LIN {X 0,Y 476.312,Z 880.73,A -85,B 0,C 180,E1 -14353.297,E2 -14353.297} C_VEL
LIN {X 0,Y 480.673,Z 862.161,A -85,B 0,C 180,E1 -14354.593,E2 -14354.593} C_VEL
LIN {X 0,Y 485.784,Z 837.994,A -85,B 0,C 180,E1 -14356.003,E2 -14356.003} C_VEL
LIN {X 0,Y 489.516,Z 817.506,A -85,B 0,C 180,E1 -14356.992,E2 -14356.992} C_VEL
LIN {X 0,Y 493.406,Z 792.396,A -85,B 0,C 180,E1 -14357.969,E2 -14357.969} C_VEL
LIN {X 0,Y 496.099,Z 770.51,A -85,B 0,C 180,E1 -14358.628,E2 -14358.628} C_VEL
LIN {X 0,Y 498.452,Z 745.206,A -85,B 0,C 180,E1 -14359.196,E2 -14359.196} C_VEL
LIN {X 0,Y 501.921,Z 674.53,A -85,B 0,C 180,E1 -14360.305,E2 -14360.305} C_VEL
LIN {X 0,Y 511.78,Z 467.818,A -85,B 0,C 180,E1 -14363.486,E2 -14363.486} C_VEL
LIN {X 0,Y 504.78,Z 456.576,A -85,B 0,C 180,E1 -14364.8,E2 -14364.8} C_VEL
LIN {X 0,Y 492.925,Z 439.35,A -85,B 0,C 180,E1 -14367.172,E2 -14367.172} C_VEL
LIN {X 0,Y 482.888,Z 425.653,A -85,B 0,C 180,E1 -14369.377,E2 -14369.377} C_VEL
LIN {X 0,Y 474.182,Z 414.504,A -85,B 0,C 180,E1 -14371.47,E2 -14371.47} C_VEL
LIN {X 0,Y 470.031,Z 409.325,A -85,B 0,C 180,E1 -14372.542,E2 -14372.542} C_VEL
LIN {X 0,Y 465.619,Z 403.891,A -85,B 0,C 180,E1 -14373.744,E2 -14373.744} C_VEL
LIN {X 0,Y 461.89,Z 399.125,A -85,B 0,C 180,E1 -14374.825,E2 -14374.825} C_VEL
LIN {X 0,Y 457.865,Z 394.726,A -85,B 0,C 180,E1 -14376.034,E2 -14376.034} C_VEL
LIN {X 0,Y 456.425,Z 392.715,A -85,B 0,C 180,E1 -14376.502,E2 -14376.502} C_VEL
LIN {X 0,Y 452.979,Z 389.244,A -85,B 0,C 180,E1 -14377.618,E2 -14377.618} C_VEL
LIN {X 0,Y 451.321,Z 386.663,A -85,B 0,C 180,E1 -14378.217,E2 -14378.217} C_VEL
LIN {X 0,Y 447.983,Z 383.799,A -85,B 0,C 180,E1 -14379.384,E2 -14379.384} C_VEL
LIN {X 0,Y 445.946,Z 380.402,A -85,B 0,C 180,E1 -14380.21,E2 -14380.21} C_VEL
LIN {X 0,Y 442.622,Z 378.058,A -85,B 0,C 180,E1 -14381.495,E2 -14381.495} C_VEL
LIN {X 0,Y 440.723,Z 374.852,A -85,B 0,C 180,E1 -14382.369,E2 -14382.369} C_VEL
LIN {X 0,Y 440.365,Z 373.869,A -85,B 0,C 180,E1 -14382.559,E2 -14382.559} C_VEL
LIN {X 0,Y 437.089,Z 372.153,A -85,B 0,C 180,E1 -14383.999,E2 -14383.999} C_VEL
LIN {X 0,Y 435.021,Z 369.435,A -85,B 0,C 180,E1 -14385.082,E2 -14385.082} C_VEL
LIN {X 0,Y 434.375,Z 367.098,A -85,B 0,C 180,E1 -14385.537,E2 -14385.537} C_VEL
LIN {X 0,Y 434.364,Z 367.103,A -85,B 0,C 180,E1 -14389.254,E2 -14389.254} C_VEL
LIN {X 0,Y 434.366,Z 367.111,A -85,B 0,C 180,E1 -14392.992,E2 -14392.992} C_VEL
LIN {X 0,Y 434.383,Z 367.122,A -85,B 0,C 180,E1 -14396.701,E2 -14396.701} C_VEL
LIN {X 0,Y 434.418,Z 367.114,A -85,B 0,C 180,E1 -14400.396,E2 -14400.396} C_VEL
LIN {X 0,Y 434.401,Z 367.104,A -85,B 0,C 180,E1 -14404.224,E2 -14404.224} C_VEL
LIN {X 0,Y 434.377,Z 367.098,A -85,B 0,C 180,E1 -14407.939,E2 -14407.939} C_VEL
LIN {X 0,Y 434.362,Z 367.095,A -85,B 0,C 180,E1 -14411.688,E2 -14411.688} C_VEL
LIN {X 0,Y 434.36,Z 367.094,A -85,B 0,C 180,E1 -14415.488,E2 -14415.488} C_VEL
LIN {X 0,Y 434.417,Z 367.337,A -85,B 0,C 180,E1 -14416.171,E2 -14416.171} C_VEL
LIN {X 0,Y 435.494,Z 370.263,A -85,B 0,C 180,E1 -14416.85,E2 -14416.85} C_VEL
LIN {X 0,Y 437.713,Z 372.671,A -85,B 0,C 180,E1 -14417.962,E2 -14417.962} C_VEL
LIN {X 0,Y 440.378,Z 374.005,A -85,B 0,C 180,E1 -14419.119,E2 -14419.119} C_VEL
LIN {X 0,Y 442.007,Z 377.269,A -85,B 0,C 180,E1 -14419.905,E2 -14419.905} C_VEL
LIN {X 0,Y 445.233,Z 380.091,A -85,B 0,C 180,E1 -14421.197,E2 -14421.197} C_VEL
LIN {X 0,Y 446.288,Z 380.829,A -85,B 0,C 180,E1 -14421.591,E2 -14421.591} C_VEL
LIN {X 0,Y 448.678,Z 384.586,A -85,B 0,C 180,E1 -14422.539,E2 -14422.539} C_VEL
LIN {X 0,Y 451.531,Z 387.353,A -85,B 0,C 180,E1 -14423.54,E2 -14423.54} C_VEL
LIN {X 0,Y 459.737,Z 397.67,A -85,B 0,C 180,E1 -14426.235,E2 -14426.235} C_VEL
LIN {X 0,Y 464.655,Z 404.165,A -85,B 0,C 180,E1 -14427.698,E2 -14427.698} C_VEL
LIN {X 0,Y 471.602,Z 413.51,A -85,B 0,C 180,E1 -14429.604,E2 -14429.604} C_VEL
LIN {X 0,Y 481.089,Z 426.79,A -85,B 0,C 180,E1 -14431.97,E2 -14431.97} C_VEL
LIN {X 0,Y 492.017,Z 443.215,A -85,B 0,C 180,E1 -14434.435,E2 -14434.435} C_VEL
LIN {X 0,Y 503.274,Z 461.442,A -85,B 0,C 180,E1 -14436.746,E2 -14436.746} C_VEL
LIN {X 0,Y 511.643,Z 476.212,A -85,B 0,C 180,E1 -14438.349,E2 -14438.349} C_VEL
LIN {X 0,Y 499.968,Z 722.479,A -85,B 0,C 180,E1 -14442.13,E2 -14442.13} C_VEL
LIN {X 0,Y 497.691,Z 766.294,A -85,B 0,C 180,E1 -14442.836,E2 -14442.836} C_VEL
LIN {X 0,Y 495.246,Z 790.201,A -85,B 0,C 180,E1 -14443.379,E2 -14443.379} C_VEL
LIN {X 0,Y 492.423,Z 811.739,A -85,B 0,C 180,E1 -14444.014,E2 -14444.014} C_VEL
LIN {X 0,Y 488.567,Z 835.485,A -85,B 0,C 180,E1 -14444.918,E2 -14444.918} C_VEL
LIN {X 0,Y 484.947,Z 854.788,A -85,B 0,C 180,E1 -14445.821,E2 -14445.821} C_VEL
LIN {X 0,Y 480.203,Z 877.436,A -85,B 0,C 180,E1 -14447.087,E2 -14447.087} C_VEL
LIN {X 0,Y 475.462,Z 897.422,A -85,B 0,C 180,E1 -14448.433,E2 -14448.433} C_VEL
LIN {X 0,Y 470.467,Z 917.266,A -85,B 0,C 180,E1 -14449.991,E2 -14449.991} C_VEL
LIN {X 0,Y 464.895,Z 937.64,A -85,B 0,C 180,E1 -14451.883,E2 -14451.883} C_VEL
LIN {X 0,Y 459.973,Z 955.021,A -85,B 0,C 180,E1 -14453.754,E2 -14453.754} C_VEL
LIN {X 0,Y 454.665,Z 973.247,A -85,B 0,C 180,E1 -14456.042,E2 -14456.042} C_VEL
LIN {X 0,Y 450.242,Z 988.386,A -85,B 0,C 180,E1 -14458.242,E2 -14458.242} C_VEL
LIN {X 0,Y 445.524,Z 1004.762,A -85,B 0,C 180,E1 -14461.003,E2 -14461.003} C_VEL
LIN {X 0,Y 441.972,Z 1017.607,A -85,B 0,C 180,E1 -14463.533,E2 -14463.533} C_VEL
LIN {X 0,Y 438.648,Z 1030.56,A -85,B 0,C 180,E1 -14466.49,E2 -14466.49} C_VEL
LIN {X 0,Y 436.221,Z 1041.033,A -85,B 0,C 180,E1 -14469.33,E2 -14469.33} C_VEL
LIN {X 0,Y 434.319,Z 1050.833,A -85,B 0,C 180,E1 -14472.447,E2 -14472.447} C_VEL
LIN {X 0,Y 433.067,Z 1058.69,A -85,B 0,C 180,E1 -14475.561,E2 -14475.561} C_VEL
LIN {X 0,Y 432.375,Z 1064.792,A -85,B 0,C 180,E1 -14478.529,E2 -14478.529} C_VEL
LIN {X 0,Y 432.028,Z 1069.722,A -85,B 0,C 180,E1 -14481.75,E2 -14481.75} C_VEL
LIN {X 0,Y 431.948,Z 1072.642,A -85,B 0,C 180,E1 -14484.494,E2 -14484.494} C_VEL
LIN {X 0,Y 431.942,Z 1074.478,A -85,B 0,C 180,E1 -14487.346,E2 -14487.346} C_VEL
LIN {X 0,Y 431.944,Z 1074.935,A -85,B 0,C 180,E1 -14490.531,E2 -14490.531} C_VEL
LIN {X 0,Y 431.947,Z 1074.097,A -85,B 0,C 180,E1 -14493.185,E2 -14493.185} C_VEL
LIN {X 0,Y 431.957,Z 1072.052,A -85,B 0,C 180,E1 -14495.979,E2 -14495.979} C_VEL
LIN {X 0,Y 432.098,Z 1067.939,A -85,B 0,C 180,E1 -14499.322,E2 -14499.322} C_VEL
LIN {X 0,Y 432.468,Z 1063.258,A -85,B 0,C 180,E1 -14502.039,E2 -14502.039} C_VEL
LIN {X 0,Y 433.263,Z 1056.581,A -85,B 0,C 180,E1 -14505.116,E2 -14505.116} C_VEL
LIN {X 0,Y 434.613,Z 1047.978,A -85,B 0,C 180,E1 -14508.233,E2 -14508.233} C_VEL
LIN {X 0,Y 436.447,Z 1038.639,A -85,B 0,C 180,E1 -14511.081,E2 -14511.081} C_VEL
LIN {X 0,Y 439.195,Z 1026.418,A -85,B 0,C 180,E1 -14514.192,E2 -14514.192} C_VEL
LIN {X 0,Y 442.123,Z 1014.703,A -85,B 0,C 180,E1 -14516.747,E2 -14516.747} C_VEL
LIN {X 0,Y 446.307,Z 998.982,A -85,B 0,C 180,E1 -14519.678,E2 -14519.678} C_VEL
LIN {X 0,Y 450.249,Z 984.69,A -85,B 0,C 180,E1 -14521.969,E2 -14521.969} C_VEL
LIN {X 0,Y 455.37,Z 966.303,A -85,B 0,C 180,E1 -14524.507,E2 -14524.507} C_VEL
LIN {X 0,Y 459.837,Z 950.082,A -85,B 0,C 180,E1 -14526.433,E2 -14526.433} C_VEL
LIN {X 0,Y 465.189,Z 930.126,A -85,B 0,C 180,E1 -14528.481,E2 -14528.481} C_VEL
LIN {X 0,Y 469.751,Z 912.077,A -85,B 0,C 180,E1 -14530.063,E2 -14530.063} C_VEL
LIN {X 0,Y 474.735,Z 891.264,A -85,B 0,C 180,E1 -14531.645,E2 -14531.645} C_VEL
LIN {X 0,Y 479.385,Z 869.689,A -85,B 0,C 180,E1 -14533.004,E2 -14533.004} C_VEL
LIN {X 0,Y 483.602,Z 848.094,A -85,B 0,C 180,E1 -14534.155,E2 -14534.155} C_VEL
LIN {X 0,Y 487.514,Z 824.79,A -85,B 0,C 180,E1 -14535.16,E2 -14535.16} C_VEL
LIN {X 0,Y 490.647,Z 802.953,A -85,B 0,C 180,E1 -14535.914,E2 -14535.914} C_VEL
LIN {X 0,Y 493.595,Z 776.73,A -85,B 0,C 180,E1 -14536.597,E2 -14536.597} C_VEL
LIN {X 0,Y 495.266,Z 754.369,A -85,B 0,C 180,E1 -14537.023,E2 -14537.023} C_VEL
LIN {X 0,Y 506.388,Z 505.867,A -85,B 0,C 180,E1 -14540.839,E2 -14540.839} C_VEL
LIN {X 0,Y 507.752,Z 473.861,A -85,B 0,C 180,E1 -14541.346,E2 -14541.346} C_VEL
LIN {X 0,Y 496.766,Z 454.506,A -85,B 0,C 180,E1 -14543.341,E2 -14543.341} C_VEL
LIN {X 0,Y 485.526,Z 436.238,A -85,B 0,C 180,E1 -14545.541,E2 -14545.541} C_VEL
LIN {X 0,Y 474.396,Z 419.479,A -85,B 0,C 180,E1 -14547.917,E2 -14547.917} C_VEL
LIN {X 0,Y 464.351,Z 405.315,A -85,B 0,C 180,E1 -14550.277,E2 -14550.277} C_VEL
LIN {X 0,Y 456.195,Z 394.492,A -85,B 0,C 180,E1 -14552.382,E2 -14552.382} C_VEL
LIN {X 0,Y 451.654,Z 388.602,A -85,B 0,C 180,E1 -14553.648,E2 -14553.648} C_VEL
LIN {X 0,Y 448.444,Z 384.751,A -85,B 0,C 180,E1 -14554.582,E2 -14554.582} C_VEL
LIN {X 0,Y 444.619,Z 379.774,A -85,B 0,C 180,E1 -14555.769,E2 -14555.769} C_VEL
LIN {X 0,Y 441.559,Z 377.023,A -85,B 0,C 180,E1 -14556.725,E2 -14556.725} C_VEL
LIN {X 0,Y 439.696,Z 373.645,A -85,B 0,C 180,E1 -14557.399,E2 -14557.399} C_VEL
LIN {X 0,Y 436.563,Z 371.7,A -85,B 0,C 180,E1 -14558.432,E2 -14558.432} C_VEL
LIN {X 0,Y 434.835,Z 368.902,A -85,B 0,C 180,E1 -14559.102,E2 -14559.102} C_VEL
LIN {X 0,Y 434.414,Z 367.107,A -85,B 0,C 180,E1 -14559.345,E2 -14559.345} C_VEL
LIN {X 0,Y 434.406,Z 367.12,A -85,B 0,C 180,E1 -14563.241,E2 -14563.241} C_VEL
LIN {X 0,Y 434.37,Z 367.098,A -85,B 0,C 180,E1 -14566.835,E2 -14566.835} C_VEL
LIN {X 0,Y 434.36,Z 367.086,A -85,B 0,C 180,E1 -14570.593,E2 -14570.593} C_VEL
LIN {X 0,Y 434.362,Z 367.096,A -85,B 0,C 180,E1 -14574.452,E2 -14574.452} C_VEL
LIN {X 0,Y 434.383,Z 367.125,A -85,B 0,C 180,E1 -14578.153,E2 -14578.153} C_VEL
LIN {X 0,Y 434.41,Z 367.084,A -85,B 0,C 180,E1 -14581.715,E2 -14581.715} C_VEL
LIN {X 0,Y 434.396,Z 367.082,A -85,B 0,C 180,E1 -14585.548,E2 -14585.548} C_VEL
LIN {X 0,Y 434.37,Z 367.117,A -85,B 0,C 180,E1 -14589.139,E2 -14589.139} C_VEL
LIN {X 0,Y 434.365,Z 367.108,A -85,B 0,C 180,E1 -14592.902,E2 -14592.902} C_VEL
LIN {X 0,Y 434.373,Z 367.087,A -85,B 0,C 180,E1 -14596.585,E2 -14596.585} C_VEL
LIN {X 0,Y 434.407,Z 367.088,A -85,B 0,C 180,E1 -14600.198,E2 -14600.198} C_VEL
LIN {X 0,Y 434.403,Z 367.369,A -85,B 0,C 180,E1 -14603.107,E2 -14603.107} C_VEL
LIN {X 0,Y 435.405,Z 370.151,A -85,B 0,C 180,E1 -14603.552,E2 -14603.552} C_VEL
LIN {X 0,Y 438.005,Z 372.837,A -85,B 0,C 180,E1 -14604.478,E2 -14604.478} C_VEL
LIN {X 0,Y 440.013,Z 374.076,A -85,B 0,C 180,E1 -14605.129,E2 -14605.129} C_VEL
LIN {X 0,Y 442.037,Z 377.566,A -85,B 0,C 180,E1 -14605.849,E2 -14605.849} C_VEL
LIN {X 0,Y 445.524,Z 380.607,A -85,B 0,C 180,E1 -14606.923,E2 -14606.923} C_VEL
LIN {X 0,Y 448.383,Z 384.646,A -85,B 0,C 180,E1 -14607.816,E2 -14607.816} C_VEL
LIN {X 0,Y 450.75,Z 386.798,A -85,B 0,C 180,E1 -14608.485,E2 -14608.485} C_VEL
LIN {X 0,Y 454.01,Z 391.044,A -85,B 0,C 180,E1 -14609.415,E2 -14609.415} C_VEL
LIN {X 0,Y 455.822,Z 392.993,A -85,B 0,C 180,E1 -14609.901,E2 -14609.901} C_VEL
LIN {X 0,Y 459.596,Z 397.562,A -85,B 0,C 180,E1 -14610.893,E2 -14610.893} C_VEL
LIN {X 0,Y 465.963,Z 405.657,A -85,B 0,C 180,E1 -14612.48,E2 -14612.48} C_VEL
LIN {X 0,Y 473.123,Z 414.677,A -85,B 0,C 180,E1 -14614.132,E2 -14614.132} C_VEL
LIN {X 0,Y 484.592,Z 430.179,A -85,B 0,C 180,E1 -14616.57,E2 -14616.57} C_VEL
LIN {X 0,Y 496.643,Z 447.502,A -85,B 0,C 180,E1 -14618.895,E2 -14618.895} C_VEL
LIN {X 0,Y 506.73,Z 463.438,A -85,B 0,C 180,E1 -14620.704,E2 -14620.704} C_VEL
LIN {X 0,Y 508.051,Z 466.028,A -85,B 0,C 180,E1 -14620.942,E2 -14620.942} C_VEL
LIN {X 0,Y 496.67,Z 717.844,A -85,B 0,C 180,E1 -14624.797,E2 -14624.797} C_VEL
LIN {X 0,Y 494.808,Z 751.173,A -85,B 0,C 180,E1 -14625.359,E2 -14625.359} C_VEL
LIN {X 0,Y 492.684,Z 773.474,A -85,B 0,C 180,E1 -14625.895,E2 -14625.895} C_VEL
LIN {X 0,Y 489.778,Z 797.274,A -85,B 0,C 180,E1 -14626.645,E2 -14626.645} C_VEL
LIN {X 0,Y 486.432,Z 818.959,A -85,B 0,C 180,E1 -14627.526,E2 -14627.526} C_VEL
LIN {X 0,Y 482.523,Z 841.197,A -85,B 0,C 180,E1 -14628.621,E2 -14628.621} C_VEL
LIN {X 0,Y 478.106,Z 862.578,A -85,B 0,C 180,E1 -14629.899,E2 -14629.899} C_VEL
LIN {X 0,Y 473.753,Z 881.913,A -85,B 0,C 180,E1 -14631.26,E2 -14631.26} C_VEL
LIN {X 0,Y 468.395,Z 903.636,A -85,B 0,C 180,E1 -14633.064,E2 -14633.064} C_VEL
LIN {X 0,Y 463.901,Z 920.654,A -85,B 0,C 180,E1 -14634.715,E2 -14634.715} C_VEL
LIN {X 0,Y 458.704,Z 939.537,A -85,B 0,C 180,E1 -14636.83,E2 -14636.83} C_VEL
LIN {X 0,Y 453.988,Z 955.906,A -85,B 0,C 180,E1 -14638.978,E2 -14638.978} C_VEL
LIN {X 0,Y 449.39,Z 972.081,A -85,B 0,C 180,E1 -14641.421,E2 -14641.421} C_VEL
LIN {X 0,Y 445.178,Z 986.714,A -85,B 0,C 180,E1 -14644.025,E2 -14644.025} C_VEL
LIN {X 0,Y 441.519,Z 1000.18,A -85,B 0,C 180,E1 -14646.793,E2 -14646.793} C_VEL
LIN {X 0,Y 438.535,Z 1011.589,A -85,B 0,C 180,E1 -14649.583,E2 -14649.583} C_VEL
LIN {X 0,Y 436.196,Z 1021.758,A -85,B 0,C 180,E1 -14652.478,E2 -14652.478} C_VEL
LIN {X 0,Y 434.361,Z 1030.763,A -85,B 0,C 180,E1 -14655.605,E2 -14655.605} C_VEL
LIN {X 0,Y 433.253,Z 1037.454,A -85,B 0,C 180,E1 -14658.417,E2 -14658.417} C_VEL
LIN {X 0,Y 432.461,Z 1043.675,A -85,B 0,C 180,E1 -14661.758,E2 -14661.758} C_VEL
LIN {X 0,Y 432.383,Z 1044.478,A -85,B 0,C 180,E1 -14662.289,E2 -14662.289} C_VEL
LIN {X 0,Y 431.252,Z 1046.049,A -85,B 0,C 180,E1 -14663.288,E2 -14663.288} C_VEL
LIN {X 0,Y 424.68,Z 1049.373,A -85,B 0,C 180,E1 -14666.043,E2 -14666.043} C_VEL
LIN {X 0,Y 424.015,Z 1050.046,A -85,B 0,C 180,E1 -14666.861,E2 -14666.861} C_VEL
LIN {X 0,Y 423.97,Z 1051.839,A -85,B 0,C 180,E1 -14670,E2 -14670} C_VEL
LIN {X 0,Y 423.952,Z 1052.046,A -85,B 0,C 180,E1 -14673.11,E2 -14673.11} C_VEL
LIN {X 0,Y 423.99,Z 1051.15,A -85,B 0,C 180,E1 -14675.82,E2 -14675.82} C_VEL
LIN {X 0,Y 424.116,Z 1048.864,A -85,B 0,C 180,E1 -14678.952,E2 -14678.952} C_VEL
LIN {X 0,Y 424.471,Z 1044.87,A -85,B 0,C 180,E1 -14682.154,E2 -14682.154} C_VEL
LIN {X 0,Y 425.153,Z 1039.888,A -85,B 0,C 180,E1 -14685.133,E2 -14685.133} C_VEL
LIN {X 0,Y 426.447,Z 1032.657,A -85,B 0,C 180,E1 -14688.453,E2 -14688.453} C_VEL
LIN {X 0,Y 428.084,Z 1025.127,A -85,B 0,C 180,E1 -14691.257,E2 -14691.257} C_VEL
LIN {X 0,Y 430.657,Z 1015.015,A -85,B 0,C 180,E1 -14694.411,E2 -14694.411} C_VEL
LIN {X 0,Y 433.776,Z 1003.834,A -85,B 0,C 180,E1 -14697.304,E2 -14697.304} C_VEL
LIN {X 0,Y 437.683,Z 990.946,A -85,B 0,C 180,E1 -14700.172,E2 -14700.172} C_VEL
LIN {X 0,Y 441.9,Z 977.282,A -85,B 0,C 180,E1 -14702.737,E2 -14702.737} C_VEL
LIN {X 0,Y 446.55,Z 962.651,A -85,B 0,C 180,E1 -14705.132,E2 -14705.132} C_VEL
LIN {X 0,Y 451.957,Z 945.292,A -85,B 0,C 180,E1 -14707.554,E2 -14707.554} C_VEL
LIN {X 0,Y 457.023,Z 928.778,A -85,B 0,C 180,E1 -14709.543,E2 -14709.543} C_VEL
LIN {X 0,Y 462.732,Z 909.231,A -85,B 0,C 180,E1 -14711.558,E2 -14711.558} C_VEL
LIN {X 0,Y 467.522,Z 891.777,A -85,B 0,C 180,E1 -14713.103,E2 -14713.103} C_VEL
LIN {X 0,Y 472.813,Z 871.108,A -85,B 0,C 180,E1 -14714.681,E2 -14714.681} C_VEL
LIN {X 0,Y 477.553,Z 850.328,A -85,B 0,C 180,E1 -14716.004,E2 -14716.004} C_VEL
LIN {X 0,Y 481.999,Z 828.767,A -85,B 0,C 180,E1 -14717.166,E2 -14717.166} C_VEL
LIN {X 0,Y 485.904,Z 806.181,A -85,B 0,C 180,E1 -14718.152,E2 -14718.152} C_VEL
LIN {X 0,Y 488.82,Z 786.379,A -85,B 0,C 180,E1 -14718.857,E2 -14718.857} C_VEL
LIN {X 0,Y 491.753,Z 761.453,A -85,B 0,C 180,E1 -14719.548,E2 -14719.548} C_VEL
LIN {X 0,Y 493.545,Z 739.017,A -85,B 0,C 180,E1 -14719.998,E2 -14719.998} C_VEL
LIN {X 0,Y 505.635,Z 494.649,A -85,B 0,C 180,E1 -14723.782,E2 -14723.782} C_VEL
LIN {X 0,Y 506.705,Z 471.513,A -85,B 0,C 180,E1 -14724.156,E2 -14724.156} C_VEL
LIN {X 0,Y 496.592,Z 455.764,A -85,B 0,C 180,E1 -14726.135,E2 -14726.135} C_VEL
LIN {X 0,Y 485.373,Z 439.786,A -85,B 0,C 180,E1 -14728.518,E2 -14728.518} C_VEL
LIN {X 0,Y 475.719,Z 426.782,A -85,B 0,C 180,E1 -14730.78,E2 -14730.78} C_VEL
LIN {X 0,Y 467.493,Z 416.348,A -85,B 0,C 180,E1 -14732.898,E2 -14732.898} C_VEL
LIN {X 0,Y 463.038,Z 410.841,A -85,B 0,C 180,E1 -14734.138,E2 -14734.138} C_VEL
LIN {X 0,Y 458.779,Z 405.565,A -85,B 0,C 180,E1 -14735.4,E2 -14735.4} C_VEL
LIN {X 0,Y 455.074,Z 401.044,A -85,B 0,C 180,E1 -14736.566,E2 -14736.566} C_VEL
LIN {X 0,Y 450.464,Z 395.877,A -85,B 0,C 180,E1 -14738.105,E2 -14738.105} C_VEL
LIN {X 0,Y 449.141,Z 394.029,A -85,B 0,C 180,E1 -14738.586,E2 -14738.586} C_VEL
LIN {X 0,Y 445.811,Z 390.841,A -85,B 0,C 180,E1 -14739.794,E2 -14739.794} C_VEL
LIN {X 0,Y 444.018,Z 387.983,A -85,B 0,C 180,E1 -14740.532,E2 -14740.532} C_VEL
LIN {X 0,Y 440.775,Z 385.427,A -85,B 0,C 180,E1 -14741.825,E2 -14741.825} C_VEL
LIN {X 0,Y 438.663,Z 381.728,A -85,B 0,C 180,E1 -14742.831,E2 -14742.831} C_VEL
LIN {X 0,Y 434.968,Z 379.222,A -85,B 0,C 180,E1 -14744.534,E2 -14744.534} C_VEL
LIN {X 0,Y 433.08,Z 376.196,A -85,B 0,C 180,E1 -14745.595,E2 -14745.595} C_VEL
LIN {X 0,Y 432.523,Z 374.865,A -85,B 0,C 180,E1 -14745.952,E2 -14745.952} C_VEL
LIN {X 0,Y 429.116,Z 373.125,A -85,B 0,C 180,E1 -14747.895,E2 -14747.895} C_VEL
LIN {X 0,Y 427.026,Z 370.28,A -85,B 0,C 180,E1 -14749.408,E2 -14749.408} C_VEL
LIN {X 0,Y 426.463,Z 368.08,A -85,B 0,C 180,E1 -14750.008,E2 -14750.008} C_VEL
LIN {X 0,Y 426.437,Z 368.086,A -85,B 0,C 180,E1 -14753.673,E2 -14753.673} C_VEL
LIN {X 0,Y 426.424,Z 368.095,A -85,B 0,C 180,E1 -14757.447,E2 -14757.447} C_VEL
LIN {X 0,Y 426.427,Z 368.106,A -85,B 0,C 180,E1 -14761.209,E2 -14761.209} C_VEL
LIN {X 0,Y 426.437,Z 368.114,A -85,B 0,C 180,E1 -14764.977,E2 -14764.977} C_VEL
LIN {X 0,Y 426.465,Z 368.095,A -85,B 0,C 180,E1 -14768.63,E2 -14768.63} C_VEL
LIN {X 0,Y 426.455,Z 368.313,A -85,B 0,C 180,E1 -14771.702,E2 -14771.702} C_VEL
LIN {X 0,Y 427.411,Z 370.977,A -85,B 0,C 180,E1 -14772.566,E2 -14772.566} C_VEL
LIN {X 0,Y 429.495,Z 373.449,A -85,B 0,C 180,E1 -14774.012,E2 -14774.012} C_VEL
LIN {X 0,Y 432.77,Z 375.179,A -85,B 0,C 180,E1 -14775.855,E2 -14775.855} C_VEL
LIN {X 0,Y 434.443,Z 378.617,A -85,B 0,C 180,E1 -14776.858,E2 -14776.858} C_VEL
LIN {X 0,Y 437.331,Z 381.042,A -85,B 0,C 180,E1 -14778.254,E2 -14778.254} C_VEL
LIN {X 0,Y 438.682,Z 381.886,A -85,B 0,C 180,E1 -14778.85,E2 -14778.85} C_VEL
LIN {X 0,Y 440.746,Z 385.354,A -85,B 0,C 180,E1 -14779.826,E2 -14779.826} C_VEL
LIN {X 0,Y 444.521,Z 388.609,A -85,B 0,C 180,E1 -14781.336,E2 -14781.336} C_VEL
LIN {X 0,Y 447.227,Z 392.486,A -85,B 0,C 180,E1 -14782.408,E2 -14782.408} C_VEL
LIN {X 0,Y 449.677,Z 394.898,A -85,B 0,C 180,E1 -14783.281,E2 -14783.281} C_VEL
LIN {X 0,Y 457.541,Z 404.981,A -85,B 0,C 180,E1 -14785.917,E2 -14785.917} C_VEL
LIN {X 0,Y 462.492,Z 411.613,A -85,B 0,C 180,E1 -14787.419,E2 -14787.419} C_VEL
LIN {X 0,Y 468.947,Z 420.397,A -85,B 0,C 180,E1 -14789.227,E2 -14789.227} C_VEL
LIN {X 0,Y 478.305,Z 433.707,A -85,B 0,C 180,E1 -14791.614,E2 -14791.614} C_VEL
LIN {X 0,Y 488.863,Z 449.818,A -85,B 0,C 180,E1 -14794.05,E2 -14794.05} C_VEL
LIN {X 0,Y 499.986,Z 468.064,A -85,B 0,C 180,E1 -14796.385,E2 -14796.385} C_VEL
LIN {X 0,Y 506.594,Z 479.918,A -85,B 0,C 180,E1 -14797.688,E2 -14797.688} C_VEL
LIN {X 0,Y 494.495,Z 726.812,A -85,B 0,C 180,E1 -14801.501,E2 -14801.501} C_VEL
LIN {X 0,Y 492.31,Z 766.561,A -85,B 0,C 180,E1 -14802.15,E2 -14802.15} C_VEL
LIN {X 0,Y 489.836,Z 790.096,A -85,B 0,C 180,E1 -14802.688,E2 -14802.688} C_VEL
LIN {X 0,Y 486.878,Z 812.003,A -85,B 0,C 180,E1 -14803.337,E2 -14803.337} C_VEL
LIN {X 0,Y 482.863,Z 835.876,A -85,B 0,C 180,E1 -14804.255,E2 -14804.255} C_VEL
LIN {X 0,Y 479.188,Z 854.851,A -85,B 0,C 180,E1 -14805.148,E2 -14805.148} C_VEL
LIN {X 0,Y 474.298,Z 877.442,A -85,B 0,C 180,E1 -14806.42,E2 -14806.42} C_VEL
LIN {X 0,Y 469.42,Z 897.339,A -85,B 0,C 180,E1 -14807.769,E2 -14807.769} C_VEL
LIN {X 0,Y 464.24,Z 917.229,A -85,B 0,C 180,E1 -14809.343,E2 -14809.343} C_VEL
LIN {X 0,Y 458.654,Z 936.961,A -85,B 0,C 180,E1 -14811.188,E2 -14811.188} C_VEL
LIN {X 0,Y 453.696,Z 953.814,A -85,B 0,C 180,E1 -14813.011,E2 -14813.011} C_VEL
LIN {X 0,Y 447.752,Z 973.418,A -85,B 0,C 180,E1 -14815.49,E2 -14815.49} C_VEL
LIN {X 0,Y 443.226,Z 988.268,A -85,B 0,C 180,E1 -14817.679,E2 -14817.679} C_VEL
LIN {X 0,Y 438.297,Z 1004.625,A -85,B 0,C 180,E1 -14820.478,E2 -14820.478} C_VEL
LIN {X 0,Y 434.57,Z 1017.461,A -85,B 0,C 180,E1 -14823.046,E2 -14823.046} C_VEL
LIN {X 0,Y 431.071,Z 1030.399,A -85,B 0,C 180,E1 -14826.051,E2 -14826.051} C_VEL
LIN {X 0,Y 428.483,Z 1040.986,A -85,B 0,C 180,E1 -14828.976,E2 -14828.976} C_VEL
LIN {X 0,Y 426.465,Z 1050.772,A -85,B 0,C 180,E1 -14832.16,E2 -14832.16} C_VEL
LIN {X 0,Y 425.154,Z 1058.506,A -85,B 0,C 180,E1 -14835.286,E2 -14835.286} C_VEL
LIN {X 0,Y 424.411,Z 1064.603,A -85,B 0,C 180,E1 -14838.31,E2 -14838.31} C_VEL
LIN {X 0,Y 424.042,Z 1069.524,A -85,B 0,C 180,E1 -14841.593,E2 -14841.593} C_VEL
LIN {X 0,Y 423.95,Z 1072.375,A -85,B 0,C 180,E1 -14844.315,E2 -14844.315} C_VEL
LIN {X 0,Y 423.945,Z 1074.203,A -85,B 0,C 180,E1 -14847.161,E2 -14847.161} C_VEL
LIN {X 0,Y 423.947,Z 1074.742,A -85,B 0,C 180,E1 -14850.405,E2 -14850.405} C_VEL
LIN {X 0,Y 423.949,Z 1073.945,A -85,B 0,C 180,E1 -14853.11,E2 -14853.11} C_VEL
LIN {X 0,Y 423.955,Z 1072.058,A -85,B 0,C 180,E1 -14855.821,E2 -14855.821} C_VEL
LIN {X 0,Y 424.076,Z 1068.332,A -85,B 0,C 180,E1 -14859.089,E2 -14859.089} C_VEL
LIN {X 0,Y 424.478,Z 1063.328,A -85,B 0,C 180,E1 -14862.102,E2 -14862.102} C_VEL
LIN {X 0,Y 425.217,Z 1057.258,A -85,B 0,C 180,E1 -14864.991,E2 -14864.991} C_VEL
LIN {X 0,Y 426.677,Z 1048.368,A -85,B 0,C 180,E1 -14868.36,E2 -14868.36} C_VEL
LIN {X 0,Y 428.526,Z 1039.3,A -85,B 0,C 180,E1 -14871.202,E2 -14871.202} C_VEL
LIN {X 0,Y 431.5,Z 1026.713,A -85,B 0,C 180,E1 -14874.506,E2 -14874.506} C_VEL
LIN {X 0,Y 434.54,Z 1015.052,A -85,B 0,C 180,E1 -14877.104,E2 -14877.104} C_VEL
LIN {X 0,Y 438.889,Z 999.45,A -85,B 0,C 180,E1 -14880.08,E2 -14880.08} C_VEL
LIN {X 0,Y 443.114,Z 984.724,A -85,B 0,C 180,E1 -14882.483,E2 -14882.483} C_VEL
LIN {X 0,Y 448.571,Z 965.947,A -85,B 0,C 180,E1 -14885.108,E2 -14885.108} C_VEL
LIN {X 0,Y 453.173,Z 949.861,A -85,B 0,C 180,E1 -14887.039,E2 -14887.039} C_VEL
LIN {X 0,Y 458.698,Z 929.968,A -85,B 0,C 180,E1 -14889.102,E2 -14889.102} C_VEL
LIN {X 0,Y 463.716,Z 910.755,A -85,B 0,C 180,E1 -14890.794,E2 -14890.794} C_VEL
LIN {X 0,Y 468.837,Z 889.947,A -85,B 0,C 180,E1 -14892.371,E2 -14892.371} C_VEL
LIN {X 0,Y 473.443,Z 869.222,A -85,B 0,C 180,E1 -14893.678,E2 -14893.678} C_VEL
LIN {X 0,Y 477.832,Z 847.403,A -85,B 0,C 180,E1 -14894.845,E2 -14894.845} C_VEL
LIN {X 0,Y 481.835,Z 824.131,A -85,B 0,C 180,E1 -14895.848,E2 -14895.848} C_VEL
LIN {X 0,Y 485.048,Z 802.306,A -85,B 0,C 180,E1 -14896.601,E2 -14896.601} C_VEL
LIN {X 0,Y 488.038,Z 776.326,A -85,B 0,C 180,E1 -14897.276,E2 -14897.276} C_VEL
LIN {X 0,Y 489.748,Z 753.945,A -85,B 0,C 180,E1 -14897.704,E2 -14897.704} C_VEL
LIN {X 0,Y 501.263,Z 505.468,A -85,B 0,C 180,E1 -14901.545,E2 -14901.545} C_VEL
LIN {X 0,Y 502.5,Z 477.419,A -85,B 0,C 180,E1 -14901.993,E2 -14901.993} C_VEL
LIN {X 0,Y 491.324,Z 457.681,A -85,B 0,C 180,E1 -14904.093,E2 -14904.093} C_VEL
LIN {X 0,Y 480.153,Z 439.521,A -85,B 0,C 180,E1 -14906.363,E2 -14906.363} C_VEL
LIN {X 0,Y 468.819,Z 422.405,A -85,B 0,C 180,E1 -14908.891,E2 -14908.891} C_VEL
LIN {X 0,Y 458.193,Z 407.553,A -85,B 0,C 180,E1 -14911.522,E2 -14911.522} C_VEL
LIN {X 0,Y 449.566,Z 396.077,A -85,B 0,C 180,E1 -14913.907,E2 -14913.907} C_VEL
LIN {X 0,Y 445.699,Z 391.494,A -85,B 0,C 180,E1 -14915.054,E2 -14915.054} C_VEL
LIN {X 0,Y 442.505,Z 387.216,A -85,B 0,C 180,E1 -14916.071,E2 -14916.071} C_VEL
LIN {X 0,Y 439.228,Z 384.03,A -85,B 0,C 180,E1 -14917.126,E2 -14917.126} C_VEL
LIN {X 0,Y 437.634,Z 381.227,A -85,B 0,C 180,E1 -14917.711,E2 -14917.711} C_VEL
LIN {X 0,Y 434.401,Z 378.872,A -85,B 0,C 180,E1 -14918.815,E2 -14918.815} C_VEL
LIN {X 0,Y 432.444,Z 375.567,A -85,B 0,C 180,E1 -14919.601,E2 -14919.601} C_VEL
LIN {X 0,Y 432.079,Z 374.761,A -85,B 0,C 180,E1 -14919.759,E2 -14919.759} C_VEL
LIN {X 0,Y 428.916,Z 372.928,A -85,B 0,C 180,E1 -14920.951,E2 -14920.951} C_VEL
LIN {X 0,Y 426.898,Z 369.924,A -85,B 0,C 180,E1 -14921.849,E2 -14921.849} C_VEL
LIN {X 0,Y 426.426,Z 368.087,A -85,B 0,C 180,E1 -14922.174,E2 -14922.174} C_VEL
LIN {X 0,Y 426.442,Z 368.074,A -85,B 0,C 180,E1 -14925.886,E2 -14925.886} C_VEL
LIN {X 0,Y 426.464,Z 368.076,A -85,B 0,C 180,E1 -14929.599,E2 -14929.599} C_VEL
LIN {X 0,Y 426.47,Z 368.105,A -85,B 0,C 180,E1 -14933.403,E2 -14933.403} C_VEL
LIN {X 0,Y 426.446,Z 368.091,A -85,B 0,C 180,E1 -14937.244,E2 -14937.244} C_VEL
LIN {X 0,Y 426.423,Z 368.071,A -85,B 0,C 180,E1 -14940.941,E2 -14940.941} C_VEL
LIN {X 0,Y 426.423,Z 368.086,A -85,B 0,C 180,E1 -14944.76,E2 -14944.76} C_VEL
LIN {X 0,Y 426.434,Z 368.114,A -85,B 0,C 180,E1 -14948.495,E2 -14948.495} C_VEL
LIN {X 0,Y 426.454,Z 368.076,A -85,B 0,C 180,E1 -14952.182,E2 -14952.182} C_VEL
LIN {X 0,Y 426.473,Z 368.07,A -85,B 0,C 180,E1 -14955.921,E2 -14955.921} C_VEL
LIN {X 0,Y 426.458,Z 368.084,A -85,B 0,C 180,E1 -14959.733,E2 -14959.733} C_VEL
LIN {X 0,Y 426.48,Z 368.249,A -85,B 0,C 180,E1 -14960.322,E2 -14960.322} C_VEL
LIN {X 0,Y 427.365,Z 370.958,A -85,B 0,C 180,E1 -14960.796,E2 -14960.796} C_VEL
LIN {X 0,Y 429.721,Z 373.581,A -85,B 0,C 180,E1 -14961.785,E2 -14961.785} C_VEL
LIN {X 0,Y 432.238,Z 375.085,A -85,B 0,C 180,E1 -14962.726,E2 -14962.726} C_VEL
LIN {X 0,Y 434.091,Z 378.452,A -85,B 0,C 180,E1 -14963.484,E2 -14963.484} C_VEL
LIN {X 0,Y 437.283,Z 381.067,A -85,B 0,C 180,E1 -14964.593,E2 -14964.593} C_VEL
LIN {X 0,Y 437.991,Z 381.856,A -85,B 0,C 180,E1 -14964.838,E2 -14964.838} C_VEL
LIN {X 0,Y 440.624,Z 385.652,A -85,B 0,C 180,E1 -14965.758,E2 -14965.758} C_VEL
LIN {X 0,Y 443.311,Z 388.033,A -85,B 0,C 180,E1 -14966.598,E2 -14966.598} C_VEL
LIN {X 0,Y 446.548,Z 392.308,A -85,B 0,C 180,E1 -14967.614,E2 -14967.614} C_VEL
LIN {X 0,Y 448.568,Z 394.354,A -85,B 0,C 180,E1 -14968.201,E2 -14968.201} C_VEL
LIN {X 0,Y 452.237,Z 398.813,A -85,B 0,C 180,E1 -14969.251,E2 -14969.251} C_VEL
LIN {X 0,Y 458.514,Z 406.657,A -85,B 0,C 180,E1 -14970.938,E2 -14970.938} C_VEL
LIN {X 0,Y 463.411,Z 412.851,A -85,B 0,C 180,E1 -14972.168,E2 -14972.168} C_VEL
LIN {X 0,Y 470.492,Z 421.952,A -85,B 0,C 180,E1 -14973.835,E2 -14973.835} C_VEL
LIN {X 0,Y 481.23,Z 436.582,A -85,B 0,C 180,E1 -14976.164,E2 -14976.164} C_VEL
LIN {X 0,Y 493.209,Z 454.026,A -85,B 0,C 180,E1 -14978.528,E2 -14978.528} C_VEL
LIN {X 0,Y 502.801,Z 469.367,A -85,B 0,C 180,E1 -14980.287,E2 -14980.287} C_VEL
LIN {X 0,Y 491.24,Z 716.754,A -85,B 0,C 180,E1 -14984.101,E2 -14984.101} C_VEL
LIN {X 0,Y 489.314,Z 750.771,A -85,B 0,C 180,E1 -14984.674,E2 -14984.674} C_VEL
LIN {X 0,Y 487.1,Z 773.465,A -85,B 0,C 180,E1 -14985.219,E2 -14985.219} C_VEL
LIN {X 0,Y 484.136,Z 797.158,A -85,B 0,C 180,E1 -14985.967,E2 -14985.967} C_VEL
LIN {X 0,Y 480.571,Z 819.588,A -85,B 0,C 180,E1 -14986.883,E2 -14986.883} C_VEL
LIN {X 0,Y 476.548,Z 841.777,A -85,B 0,C 180,E1 -14987.985,E2 -14987.985} C_VEL
LIN {X 0,Y 471.793,Z 863.976,A -85,B 0,C 180,E1 -14989.33,E2 -14989.33} C_VEL
LIN {X 0,Y 467.112,Z 884.074,A -85,B 0,C 180,E1 -14990.77,E2 -14990.77} C_VEL
LIN {X 0,Y 461.787,Z 904.731,A -85,B 0,C 180,E1 -14992.523,E2 -14992.523} C_VEL
LIN {X 0,Y 457.153,Z 921.671,A -85,B 0,C 180,E1 -14994.192,E2 -14994.192} C_VEL
LIN {X 0,Y 451.475,Z 941.415,A -85,B 0,C 180,E1 -14996.456,E2 -14996.456} C_VEL
LIN {X 0,Y 447.009,Z 956.39,A -85,B 0,C 180,E1 -14998.457,E2 -14998.457} C_VEL
LIN {X 0,Y 442.252,Z 972.428,A -85,B 0,C 180,E1 -15000.916,E2 -15000.916} C_VEL
LIN {X 0,Y 437.937,Z 986.804,A -85,B 0,C 180,E1 -15003.51,E2 -15003.51} C_VEL
LIN {X 0,Y 434.034,Z 1000.496,A -85,B 0,C 180,E1 -15006.369,E2 -15006.369} C_VEL
LIN {X 0,Y 430.845,Z 1012.145,A -85,B 0,C 180,E1 -15009.273,E2 -15009.273} C_VEL
LIN {X 0,Y 428.321,Z 1022.647,A -85,B 0,C 180,E1 -15012.333,E2 -15012.333} C_VEL
LIN {X 0,Y 426.445,Z 1031.387,A -85,B 0,C 180,E1 -15015.47,E2 -15015.47} C_VEL
LIN {X 0,Y 425.213,Z 1038.613,A -85,B 0,C 180,E1 -15018.608,E2 -15018.608} C_VEL
LIN {X 0,Y 424.455,Z 1044.329,A -85,B 0,C 180,E1 -15021.875,E2 -15021.875} C_VEL
LIN {X 0,Y 424.131,Z 1048.056,A -85,B 0,C 180,E1 -15024.725,E2 -15024.725} C_VEL
LIN {X 0,Y 424.015,Z 1050.046,A -85,B 0,C 180,E1 -15026.861,E2 -15026.861} C_VEL
LIN {X 0,Y 422.997,Z 1050.856,A -85,B 0,C 180,E1 -15027.896,E2 -15027.896} C_VEL
LIN {X 0,Y 416.589,Z 1052.175,A -85,B 0,C 180,E1 -15030.745,E2 -15030.745} C_VEL
LIN {X 0,Y 415.945,Z 1052.314,A -85,B 0,C 180,E1 -15031.587,E2 -15031.587} C_VEL
LIN {X 0,Y 415.972,Z 1051.818,A -85,B 0,C 180,E1 -15034.964,E2 -15034.964} C_VEL
LIN {X 0,Y 416.052,Z 1050.071,A -85,B 0,C 180,E1 -15037.874,E2 -15037.874} C_VEL
LIN {X 0,Y 416.291,Z 1047.175,A -85,B 0,C 180,E1 -15040.798,E2 -15040.798} C_VEL
LIN {X 0,Y 416.939,Z 1042.004,A -85,B 0,C 180,E1 -15044.335,E2 -15044.335} C_VEL
LIN {X 0,Y 417.92,Z 1036.341,A -85,B 0,C 180,E1 -15047.258,E2 -15047.258} C_VEL
LIN {X 0,Y 419.71,Z 1028.169,A -85,B 0,C 180,E1 -15050.646,E2 -15050.646} C_VEL
LIN {X 0,Y 421.935,Z 1019.336,A -85,B 0,C 180,E1 -15053.609,E2 -15053.609} C_VEL
LIN {X 0,Y 425.07,Z 1008.503,A -85,B 0,C 180,E1 -15056.698,E2 -15056.698} C_VEL
LIN {X 0,Y 428.861,Z 996.143,A -85,B 0,C 180,E1 -15059.622,E2 -15059.622} C_VEL
LIN {X 0,Y 433.239,Z 982.686,A -85,B 0,C 180,E1 -15062.374,E2 -15062.374} C_VEL
LIN {X 0,Y 438.22,Z 967.455,A -85,B 0,C 180,E1 -15065.001,E2 -15065.001} C_VEL
LIN {X 0,Y 443.075,Z 952.695,A -85,B 0,C 180,E1 -15067.214,E2 -15067.214} C_VEL
LIN {X 0,Y 449.039,Z 934.034,A -85,B 0,C 180,E1 -15069.605,E2 -15069.605} C_VEL
LIN {X 0,Y 454.325,Z 916.902,A -85,B 0,C 180,E1 -15071.487,E2 -15071.487} C_VEL
LIN {X 0,Y 460.35,Z 896.166,A -85,B 0,C 180,E1 -15073.428,E2 -15073.428} C_VEL
LIN {X 0,Y 465.245,Z 877.922,A -85,B 0,C 180,E1 -15074.884,E2 -15074.884} C_VEL
LIN {X 0,Y 470.527,Z 856.532,A -85,B 0,C 180,E1 -15076.342,E2 -15076.342} C_VEL
LIN {X 0,Y 475.1,Z 835.421,A -85,B 0,C 180,E1 -15077.532,E2 -15077.532} C_VEL
LIN {X 0,Y 479.346,Z 813.232,A -85,B 0,C 180,E1 -15078.582,E2 -15078.582} C_VEL
LIN {X 0,Y 482.959,Z 790.065,A -85,B 0,C 180,E1 -15079.448,E2 -15079.448} C_VEL
LIN {X 0,Y 485.749,Z 768.223,A -85,B 0,C 180,E1 -15080.094,E2 -15080.094} C_VEL
LIN {X 0,Y 488.106,Z 742.445,A -85,B 0,C 180,E1 -15080.649,E2 -15080.649} C_VEL
LIN {X 0,Y 500.063,Z 509.034,A -85,B 0,C 180,E1 -15084.292,E2 -15084.292} C_VEL
LIN {X 0,Y 501.723,Z 475.289,A -85,B 0,C 180,E1 -15084.833,E2 -15084.833} C_VEL
LIN {X 0,Y 491.043,Z 458.951,A -85,B 0,C 180,E1 -15086.996,E2 -15086.996} C_VEL
LIN {X 0,Y 480.225,Z 443.43,A -85,B 0,C 180,E1 -15089.397,E2 -15089.397} C_VEL
LIN {X 0,Y 469.661,Z 429.257,A -85,B 0,C 180,E1 -15092.002,E2 -15092.002} C_VEL
LIN {X 0,Y 460.98,Z 418.3,A -85,B 0,C 180,E1 -15094.394,E2 -15094.394} C_VEL
LIN {X 0,Y 456.288,Z 412.56,A -85,B 0,C 180,E1 -15095.809,E2 -15095.809} C_VEL
LIN {X 0,Y 451.936,Z 407.223,A -85,B 0,C 180,E1 -15097.221,E2 -15097.221} C_VEL
LIN {X 0,Y 448.305,Z 403.012,A -85,B 0,C 180,E1 -15098.475,E2 -15098.475} C_VEL
LIN {X 0,Y 447.158,Z 401.478,A -85,B 0,C 180,E1 -15098.899,E2 -15098.899} C_VEL
LIN {X 0,Y 443.662,Z 397.874,A -85,B 0,C 180,E1 -15100.207,E2 -15100.207} C_VEL
LIN {X 0,Y 442.109,Z 395.52,A -85,B 0,C 180,E1 -15100.856,E2 -15100.856} C_VEL
LIN {X 0,Y 438.805,Z 392.613,A -85,B 0,C 180,E1 -15102.221,E2 -15102.221} C_VEL
LIN {X 0,Y 436.709,Z 389.232,A -85,B 0,C 180,E1 -15103.232,E2 -15103.232} C_VEL
LIN {X 0,Y 433.255,Z 386.635,A -85,B 0,C 180,E1 -15104.883,E2 -15104.883} C_VEL
LIN {X 0,Y 431.273,Z 383.204,A -85,B 0,C 180,E1 -15106.047,E2 -15106.047} C_VEL
LIN {X 0,Y 430.836,Z 382.617,A -85,B 0,C 180,E1 -15106.307,E2 -15106.307} C_VEL
LIN {X 0,Y 427.55,Z 380.636,A -85,B 0,C 180,E1 -15108.26,E2 -15108.26} C_VEL
LIN {X 0,Y 425.626,Z 377.822,A -85,B 0,C 180,E1 -15109.715,E2 -15109.715} C_VEL
LIN {X 0,Y 424.917,Z 375.931,A -85,B 0,C 180,E1 -15110.382,E2 -15110.382} C_VEL
LIN {X 0,Y 420.979,Z 373.898,A -85,B 0,C 180,E1 -15114.138,E2 -15114.138} C_VEL
LIN {X 0,Y 418.688,Z 370.127,A -85,B 0,C 180,E1 -15119.453,E2 -15119.453} C_VEL
LIN {X 0,Y 418.612,Z 369.749,A -85,B 0,C 180,E1 -15120.821,E2 -15120.821} C_VEL
LIN {X 0,Y 418.818,Z 370.545,A -85,B 0,C 180,E1 -15123.011,E2 -15123.011} C_VEL
LIN {X 0,Y 423.403,Z 375.494,A -85,B 0,C 180,E1 -15130.064,E2 -15130.064} C_VEL
LIN {X 0,Y 425.089,Z 376.181,A -85,B 0,C 180,E1 -15131.43,E2 -15131.43} C_VEL
LIN {X 0,Y 426.592,Z 379.531,A -85,B 0,C 180,E1 -15132.728,E2 -15132.728} C_VEL
LIN {X 0,Y 429.411,Z 381.997,A -85,B 0,C 180,E1 -15134.565,E2 -15134.565} C_VEL
LIN {X 0,Y 431.26,Z 383.048,A -85,B 0,C 180,E1 -15135.602,E2 -15135.602} C_VEL
LIN {X 0,Y 433.226,Z 386.626,A -85,B 0,C 180,E1 -15136.768,E2 -15136.768} C_VEL
LIN {X 0,Y 436.396,Z 389.06,A -85,B 0,C 180,E1 -15138.295,E2 -15138.295} C_VEL
LIN {X 0,Y 437.075,Z 389.746,A -85,B 0,C 180,E1 -15138.611,E2 -15138.611} C_VEL
LIN {X 0,Y 439.638,Z 393.534,A -85,B 0,C 180,E1 -15139.809,E2 -15139.809} C_VEL
LIN {X 0,Y 442.695,Z 396.176,A -85,B 0,C 180,E1 -15141.047,E2 -15141.047} C_VEL
LIN {X 0,Y 445.617,Z 400.199,A -85,B 0,C 180,E1 -15142.215,E2 -15142.215} C_VEL
LIN {X 0,Y 448.034,Z 402.698,A -85,B 0,C 180,E1 -15143.093,E2 -15143.093} C_VEL
LIN {X 0,Y 455.36,Z 412.285,A -85,B 0,C 180,E1 -15145.596,E2 -15145.596} C_VEL
LIN {X 0,Y 460.534,Z 419.318,A -85,B 0,C 180,E1 -15147.196,E2 -15147.196} C_VEL
LIN {X 0,Y 466.618,Z 427.734,A -85,B 0,C 180,E1 -15148.931,E2 -15148.931} C_VEL
LIN {X 0,Y 475.649,Z 440.785,A -85,B 0,C 180,E1 -15151.281,E2 -15151.281} C_VEL
LIN {X 0,Y 485.731,Z 456.417,A -85,B 0,C 180,E1 -15153.66,E2 -15153.66} C_VEL
LIN {X 0,Y 496.408,Z 474.181,A -85,B 0,C 180,E1 -15155.956,E2 -15155.956} C_VEL
LIN {X 0,Y 501.607,Z 483.771,A -85,B 0,C 180,E1 -15157.016,E2 -15157.016} C_VEL
LIN {X 0,Y 489.101,Z 730.776,A -85,B 0,C 180,E1 -15160.852,E2 -15160.852} C_VEL
LIN {X 0,Y 486.969,Z 767.159,A -85,B 0,C 180,E1 -15161.457,E2 -15161.457} C_VEL
LIN {X 0,Y 484.48,Z 790.135,A -85,B 0,C 180,E1 -15161.985,E2 -15161.985} C_VEL
LIN {X 0,Y 481.316,Z 812.88,A -85,B 0,C 180,E1 -15162.664,E2 -15162.664} C_VEL
LIN {X 0,Y 477.335,Z 835.692,A -85,B 0,C 180,E1 -15163.55,E2 -15163.55} C_VEL
LIN {X 0,Y 473.495,Z 854.917,A -85,B 0,C 180,E1 -15164.458,E2 -15164.458} C_VEL
LIN {X 0,Y 468.282,Z 878.153,A -85,B 0,C 180,E1 -15165.782,E2 -15165.782} C_VEL
LIN {X 0,Y 463.407,Z 897.39,A -85,B 0,C 180,E1 -15167.098,E2 -15167.098} C_VEL
LIN {X 0,Y 457.88,Z 917.929,A -85,B 0,C 180,E1 -15168.739,E2 -15168.739} C_VEL
LIN {X 0,Y 451.979,Z 937.935,A -85,B 0,C 180,E1 -15170.645,E2 -15170.645} C_VEL
LIN {X 0,Y 446.652,Z 955.402,A -85,B 0,C 180,E1 -15172.57,E2 -15172.57} C_VEL
LIN {X 0,Y 441.063,Z 973.032,A -85,B 0,C 180,E1 -15174.843,E2 -15174.843} C_VEL
LIN {X 0,Y 436.255,Z 988.151,A -85,B 0,C 180,E1 -15177.098,E2 -15177.098} C_VEL
LIN {X 0,Y 431.109,Z 1004.489,A -85,B 0,C 180,E1 -15179.935,E2 -15179.935} C_VEL
LIN {X 0,Y 427.269,Z 1017.077,A -85,B 0,C 180,E1 -15182.491,E2 -15182.491} C_VEL
LIN {X 0,Y 423.524,Z 1030.24,A -85,B 0,C 180,E1 -15185.597,E2 -15185.597} C_VEL
LIN {X 0,Y 420.817,Z 1040.699,A -85,B 0,C 180,E1 -15188.536,E2 -15188.536} C_VEL
LIN {X 0,Y 418.67,Z 1050.475,A -85,B 0,C 180,E1 -15191.768,E2 -15191.768} C_VEL
LIN {X 0,Y 417.246,Z 1058.322,A -85,B 0,C 180,E1 -15195,E2 -15195} C_VEL
LIN {X 0,Y 416.452,Z 1064.415,A -85,B 0,C 180,E1 -15198.084,E2 -15198.084} C_VEL
LIN {X 0,Y 416.053,Z 1069.326,A -85,B 0,C 180,E1 -15201.431,E2 -15201.431} C_VEL
LIN {X 0,Y 415.953,Z 1072.173,A -85,B 0,C 180,E1 -15204.205,E2 -15204.205} C_VEL
LIN {X 0,Y 415.947,Z 1073.996,A -85,B 0,C 180,E1 -15207.106,E2 -15207.106} C_VEL
LIN {X 0,Y 415.951,Z 1074.526,A -85,B 0,C 180,E1 -15210.413,E2 -15210.413} C_VEL
LIN {X 0,Y 415.951,Z 1073.724,A -85,B 0,C 180,E1 -15213.169,E2 -15213.169} C_VEL
LIN {X 0,Y 415.958,Z 1071.831,A -85,B 0,C 180,E1 -15215.933,E2 -15215.933} C_VEL
LIN {X 0,Y 416.09,Z 1068.093,A -85,B 0,C 180,E1 -15219.265,E2 -15219.265} C_VEL
LIN {X 0,Y 416.522,Z 1063.082,A -85,B 0,C 180,E1 -15222.336,E2 -15222.336} C_VEL
LIN {X 0,Y 417.312,Z 1057.005,A -85,B 0,C 180,E1 -15225.282,E2 -15225.282} C_VEL
LIN {X 0,Y 418.828,Z 1048.271,A -85,B 0,C 180,E1 -15228.657,E2 -15228.657} C_VEL
LIN {X 0,Y 420.717,Z 1039.492,A -85,B 0,C 180,E1 -15231.469,E2 -15231.469} C_VEL
LIN {X 0,Y 423.668,Z 1027.59,A -85,B 0,C 180,E1 -15234.692,E2 -15234.692} C_VEL
LIN {X 0,Y 426.974,Z 1015.4,A -85,B 0,C 180,E1 -15237.473,E2 -15237.473} C_VEL
LIN {X 0,Y 431.27,Z 1000.7,A -85,B 0,C 180,E1 -15240.36,E2 -15240.36} C_VEL
LIN {X 0,Y 435.756,Z 985.622,A -85,B 0,C 180,E1 -15242.878,E2 -15242.878} C_VEL
LIN {X 0,Y 440.916,Z 968.695,A -85,B 0,C 180,E1 -15245.329,E2 -15245.329} C_VEL
LIN {X 0,Y 446.124,Z 951.105,A -85,B 0,C 180,E1 -15247.494,E2 -15247.494} C_VEL
LIN {X 0,Y 451.673,Z 932.049,A -85,B 0,C 180,E1 -15249.528,E2 -15249.528} C_VEL
LIN {X 0,Y 457.131,Z 911.839,A -85,B 0,C 180,E1 -15251.343,E2 -15251.343} C_VEL
LIN {X 0,Y 462.399,Z 891.244,A -85,B 0,C 180,E1 -15252.934,E2 -15252.934} C_VEL
LIN {X 0,Y 467.35,Z 869.768,A -85,B 0,C 180,E1 -15254.31,E2 -15254.31} C_VEL
LIN {X 0,Y 471.676,Z 848.949,A -85,B 0,C 180,E1 -15255.438,E2 -15255.438} C_VEL
LIN {X 0,Y 476.012,Z 824.836,A -85,B 0,C 180,E1 -15256.499,E2 -15256.499} C_VEL
LIN {X 0,Y 479.336,Z 802.967,A -85,B 0,C 180,E1 -15257.262,E2 -15257.262} C_VEL
LIN {X 0,Y 482.499,Z 776.475,A -85,B 0,C 180,E1 -15257.959,E2 -15257.959} C_VEL
LIN {X 0,Y 484.261,Z 754.165,A -85,B 0,C 180,E1 -15258.389,E2 -15258.389} C_VEL
LIN {X 0,Y 496.168,Z 506.014,A -85,B 0,C 180,E1 -15262.251,E2 -15262.251} C_VEL
LIN {X 0,Y 497.264,Z 480.875,A -85,B 0,C 180,E1 -15262.663,E2 -15262.663} C_VEL
LIN {X 0,Y 485.976,Z 460.861,A -85,B 0,C 180,E1 -15264.859,E2 -15264.859} C_VEL
LIN {X 0,Y 475.949,Z 444.657,A -85,B 0,C 180,E1 -15266.964,E2 -15266.964} C_VEL
LIN {X 0,Y 465.74,Z 428.971,A -85,B 0,C 180,E1 -15269.308,E2 -15269.308} C_VEL
LIN {X 0,Y 455.376,Z 414.304,A -85,B 0,C 180,E1 -15271.937,E2 -15271.937} C_VEL
LIN {X 0,Y 446.885,Z 402.869,A -85,B 0,C 180,E1 -15274.345,E2 -15274.345} C_VEL
LIN {X 0,Y 440.971,Z 395.228,A -85,B 0,C 180,E1 -15276.196,E2 -15276.196} C_VEL
LIN {X 0,Y 436.919,Z 391.036,A -85,B 0,C 180,E1 -15277.531,E2 -15277.531} C_VEL
LIN {X 0,Y 435.592,Z 388.754,A -85,B 0,C 180,E1 -15278.027,E2 -15278.027} C_VEL
LIN {X 0,Y 432.26,Z 386.031,A -85,B 0,C 180,E1 -15279.202,E2 -15279.202} C_VEL
LIN {X 0,Y 429.94,Z 382.324,A -85,B 0,C 180,E1 -15280.151,E2 -15280.151} C_VEL
LIN {X 0,Y 426.729,Z 379.982,A -85,B 0,C 180,E1 -15281.417,E2 -15281.417} C_VEL
LIN {X 0,Y 424.725,Z 376.641,A -85,B 0,C 180,E1 -15282.356,E2 -15282.356} C_VEL
LIN {X 0,Y 424.263,Z 375.798,A -85,B 0,C 180,E1 -15282.584,E2 -15282.584} C_VEL
LIN {X 0,Y 420.826,Z 373.806,A -85,B 0,C 180,E1 -15284.143,E2 -15284.143} C_VEL
LIN {X 0,Y 419.073,Z 371.165,A -85,B 0,C 180,E1 -15285.103,E2 -15285.103} C_VEL
LIN {X 0,Y 418.534,Z 369.058,A -85,B 0,C 180,E1 -15285.539,E2 -15285.539} C_VEL
LIN {X 0,Y 418.524,Z 369.067,A -85,B 0,C 180,E1 -15289.399,E2 -15289.399} C_VEL
LIN {X 0,Y 418.506,Z 369.102,A -85,B 0,C 180,E1 -15293.139,E2 -15293.139} C_VEL
LIN {X 0,Y 418.486,Z 369.072,A -85,B 0,C 180,E1 -15296.85,E2 -15296.85} C_VEL
LIN {X 0,Y 418.483,Z 369.059,A -85,B 0,C 180,E1 -15300.685,E2 -15300.685} C_VEL
LIN {X 0,Y 418.489,Z 369.078,A -85,B 0,C 180,E1 -15304.522,E2 -15304.522} C_VEL
LIN {X 0,Y 418.51,Z 369.095,A -85,B 0,C 180,E1 -15308.242,E2 -15308.242} C_VEL
LIN {X 0,Y 418.525,Z 369.06,A -85,B 0,C 180,E1 -15311.996,E2 -15311.996} C_VEL
LIN {X 0,Y 418.516,Z 369.061,A -85,B 0,C 180,E1 -15315.673,E2 -15315.673} C_VEL
LIN {X 0,Y 418.514,Z 369.269,A -85,B 0,C 180,E1 -15316.929,E2 -15316.929} C_VEL
LIN {X 0,Y 419.428,Z 371.93,A -85,B 0,C 180,E1 -15317.527,E2 -15317.527} C_VEL
LIN {X 0,Y 421.919,Z 374.717,A -85,B 0,C 180,E1 -15318.802,E2 -15318.802} C_VEL
LIN {X 0,Y 424.495,Z 375.974,A -85,B 0,C 180,E1 -15319.935,E2 -15319.935} C_VEL
LIN {X 0,Y 426.155,Z 379.317,A -85,B 0,C 180,E1 -15320.75,E2 -15320.75} C_VEL
LIN {X 0,Y 428.96,Z 381.799,A -85,B 0,C 180,E1 -15321.898,E2 -15321.898} C_VEL
LIN {X 0,Y 430.281,Z 382.728,A -85,B 0,C 180,E1 -15322.402,E2 -15322.402} C_VEL
LIN {X 0,Y 432.629,Z 386.398,A -85,B 0,C 180,E1 -15323.352,E2 -15323.352} C_VEL
LIN {X 0,Y 435.876,Z 389.234,A -85,B 0,C 180,E1 -15324.497,E2 -15324.497} C_VEL
LIN {X 0,Y 438.94,Z 393.394,A -85,B 0,C 180,E1 -15325.574,E2 -15325.574} C_VEL
LIN {X 0,Y 441.207,Z 395.549,A -85,B 0,C 180,E1 -15326.299,E2 -15326.299} C_VEL
LIN {X 0,Y 444.82,Z 400.05,A -85,B 0,C 180,E1 -15327.44,E2 -15327.44} C_VEL
LIN {X 0,Y 446.499,Z 401.996,A -85,B 0,C 180,E1 -15327.943,E2 -15327.943} C_VEL
LIN {X 0,Y 451.267,Z 407.869,A -85,B 0,C 180,E1 -15329.32,E2 -15329.32} C_VEL
LIN {X 0,Y 456.246,Z 414.141,A -85,B 0,C 180,E1 -15330.67,E2 -15330.67} C_VEL
LIN {X 0,Y 463.604,Z 423.42,A -85,B 0,C 180,E1 -15332.519,E2 -15332.519} C_VEL
LIN {X 0,Y 474.453,Z 438.155,A -85,B 0,C 180,E1 -15335.013,E2 -15335.013} C_VEL
LIN {X 0,Y 486.127,Z 454.989,A -85,B 0,C 180,E1 -15337.438,E2 -15337.438} C_VEL
LIN {X 0,Y 497.481,Z 472.781,A -85,B 0,C 180,E1 -15339.602,E2 -15339.602} C_VEL
LIN {X 0,Y 494.245,Z 540.572,A -85,B 0,C 180,E1 -15340.671,E2 -15340.671} C_VEL
LIN {X 0,Y 484.404,Z 743.34,A -85,B 0,C 180,E1 -15343.841,E2 -15343.841} C_VEL
LIN {X 0,Y 481.987,Z 769.926,A -85,B 0,C 180,E1 -15344.432,E2 -15344.432} C_VEL
LIN {X 0,Y 479.3,Z 791.582,A -85,B 0,C 180,E1 -15345.087,E2 -15345.087} C_VEL
LIN {X 0,Y 475.451,Z 816.4,A -85,B 0,C 180,E1 -15346.052,E2 -15346.052} C_VEL
LIN {X 0,Y 471.704,Z 836.768,A -85,B 0,C 180,E1 -15347.039,E2 -15347.039} C_VEL
LIN {X 0,Y 466.993,Z 859.147,A -85,B 0,C 180,E1 -15348.332,E2 -15348.332} C_VEL
LIN {X 0,Y 462.092,Z 879.669,A -85,B 0,C 180,E1 -15349.767,E2 -15349.767} C_VEL
LIN {X 0,Y 456.702,Z 900.554,A -85,B 0,C 180,E1 -15351.474,E2 -15351.474} C_VEL
LIN {X 0,Y 451.337,Z 919.524,A -85,B 0,C 180,E1 -15353.319,E2 -15353.319} C_VEL
LIN {X 0,Y 446.028,Z 937.684,A -85,B 0,C 180,E1 -15355.359,E2 -15355.359} C_VEL
LIN {X 0,Y 440.715,Z 954.826,A -85,B 0,C 180,E1 -15357.627,E2 -15357.627} C_VEL
LIN {X 0,Y 436.139,Z 969.53,A -85,B 0,C 180,E1 -15359.862,E2 -15359.862} C_VEL
LIN {X 0,Y 431.22,Z 985.321,A -85,B 0,C 180,E1 -15362.67,E2 -15362.67} C_VEL
LIN {X 0,Y 427.607,Z 997.226,A -85,B 0,C 180,E1 -15365.132,E2 -15365.132} C_VEL
LIN {X 0,Y 423.882,Z 1010.18,A -85,B 0,C 180,E1 -15368.263,E2 -15368.263} C_VEL
LIN {X 0,Y 421.31,Z 1019.806,A -85,B 0,C 180,E1 -15371.026,E2 -15371.026} C_VEL
LIN {X 0,Y 419.123,Z 1029.244,A -85,B 0,C 180,E1 -15374.219,E2 -15374.219} C_VEL
LIN {X 0,Y 417.622,Z 1036.803,A -85,B 0,C 180,E1 -15377.416,E2 -15377.416} C_VEL
LIN {X 0,Y 416.736,Z 1042.66,A -85,B 0,C 180,E1 -15380.471,E2 -15380.471} C_VEL
LIN {X 0,Y 416.211,Z 1047.36,A -85,B 0,C 180,E1 -15383.794,E2 -15383.794} C_VEL
LIN {X 0,Y 416.029,Z 1050.081,A -85,B 0,C 180,E1 -15386.555,E2 -15386.555} C_VEL
LIN {X 0,Y 415.964,Z 1051.822,A -85,B 0,C 180,E1 -15389.449,E2 -15389.449} C_VEL
LIN {X 0,Y 415.945,Z 1052.314,A -85,B 0,C 180,E1 -15391.587,E2 -15391.587} C_VEL
LIN {X 0,Y 414.951,Z 1052.399,A -85,B 0,C 180,E1 -15392.648,E2 -15392.648} C_VEL
LIN {X 0,Y 408.628,Z 1051.776,A -85,B 0,C 180,E1 -15395.56,E2 -15395.56} C_VEL
LIN {X 0,Y 408.018,Z 1051.383,A -85,B 0,C 180,E1 -15396.417,E2 -15396.417} C_VEL
LIN {X 0,Y 408.201,Z 1048.616,A -85,B 0,C 180,E1 -15399.873,E2 -15399.873} C_VEL
LIN {X 0,Y 408.619,Z 1044.904,A -85,B 0,C 180,E1 -15402.866,E2 -15402.866} C_VEL
LIN {X 0,Y 409.527,Z 1039.483,A -85,B 0,C 180,E1 -15406.161,E2 -15406.161} C_VEL
LIN {X 0,Y 411.021,Z 1032.276,A -85,B 0,C 180,E1 -15409.468,E2 -15409.468} C_VEL
LIN {X 0,Y 413.044,Z 1024.314,A -85,B 0,C 180,E1 -15412.488,E2 -15412.488} C_VEL
LIN {X 0,Y 416.061,Z 1013.749,A -85,B 0,C 180,E1 -15415.784,E2 -15415.784} C_VEL
LIN {X 0,Y 419.272,Z 1003.511,A -85,B 0,C 180,E1 -15418.487,E2 -15418.487} C_VEL
LIN {X 0,Y 423.933,Z 989.517,A -85,B 0,C 180,E1 -15421.629,E2 -15421.629} C_VEL
LIN {X 0,Y 428.3,Z 976.696,A -85,B 0,C 180,E1 -15424.076,E2 -15424.076} C_VEL
LIN {X 0,Y 433.702,Z 961.072,A -85,B 0,C 180,E1 -15426.664,E2 -15426.664} C_VEL
LIN {X 0,Y 439.234,Z 944.626,A -85,B 0,C 180,E1 -15428.968,E2 -15428.968} C_VEL
LIN {X 0,Y 445.194,Z 926.627,A -85,B 0,C 180,E1 -15431.153,E2 -15431.153} C_VEL
LIN {X 0,Y 450.958,Z 907.89,A -85,B 0,C 180,E1 -15433.072,E2 -15433.072} C_VEL
LIN {X 0,Y 456.331,Z 889.523,A -85,B 0,C 180,E1 -15434.697,E2 -15434.697} C_VEL
LIN {X 0,Y 461.985,Z 868.244,A -85,B 0,C 180,E1 -15436.293,E2 -15436.293} C_VEL
LIN {X 0,Y 466.58,Z 849.267,A -85,B 0,C 180,E1 -15437.493,E2 -15437.493} C_VEL
LIN {X 0,Y 471.476,Z 826.43,A -85,B 0,C 180,E1 -15438.712,E2 -15438.712} C_VEL
LIN {X 0,Y 475.423,Z 804.541,A -85,B 0,C 180,E1 -15439.652,E2 -15439.652} C_VEL
LIN {X 0,Y 478.794,Z 782.599,A -85,B 0,C 180,E1 -15440.416,E2 -15440.416} C_VEL
LIN {X 0,Y 481.612,Z 758.204,A -85,B 0,C 180,E1 -15441.057,E2 -15441.057} C_VEL
LIN {X 0,Y 483.399,Z 735.982,A -85,B 0,C 180,E1 -15441.488,E2 -15441.488} C_VEL
LIN {X 0,Y 496.618,Z 485.293,A -85,B 0,C 180,E1 -15445.404,E2 -15445.404} C_VEL
LIN {X 0,Y 496.914,Z 479.493,A -85,B 0,C 180,E1 -15445.498,E2 -15445.498} C_VEL
LIN {X 0,Y 486.438,Z 463.357,A -85,B 0,C 180,E1 -15447.694,E2 -15447.694} C_VEL
LIN {X 0,Y 476.625,Z 449.248,A -85,B 0,C 180,E1 -15449.943,E2 -15449.943} C_VEL
LIN {X 0,Y 466.885,Z 436.027,A -85,B 0,C 180,E1 -15452.411,E2 -15452.411} C_VEL
LIN {X 0,Y 458.438,Z 425.238,A -85,B 0,C 180,E1 -15454.795,E2 -15454.795} C_VEL
LIN {X 0,Y 454.01,Z 419.728,A -85,B 0,C 180,E1 -15456.163,E2 -15456.163} C_VEL
LIN {X 0,Y 449.722,Z 414.447,A -85,B 0,C 180,E1 -15457.585,E2 -15457.585} C_VEL
LIN {X 0,Y 446.007,Z 409.892,A -85,B 0,C 180,E1 -15458.911,E2 -15458.911} C_VEL
LIN {X 0,Y 441.392,Z 404.67,A -85,B 0,C 180,E1 -15460.686,E2 -15460.686} C_VEL
LIN {X 0,Y 440.218,Z 403.028,A -85,B 0,C 180,E1 -15461.184,E2 -15461.184} C_VEL
LIN {X 0,Y 436.857,Z 399.787,A -85,B 0,C 180,E1 -15462.621,E2 -15462.621} C_VEL
LIN {X 0,Y 435.195,Z 396.978,A -85,B 0,C 180,E1 -15463.447,E2 -15463.447} C_VEL
LIN {X 0,Y 431.677,Z 394.181,A -85,B 0,C 180,E1 -15465.17,E2 -15465.17} C_VEL
LIN {X 0,Y 429.405,Z 390.424,A -85,B 0,C 180,E1 -15466.535,E2 -15466.535} C_VEL
LIN {X 0,Y 426.191,Z 388.334,A -85,B 0,C 180,E1 -15468.497,E2 -15468.497} C_VEL
LIN {X 0,Y 424.238,Z 385.362,A -85,B 0,C 180,E1 -15470.024,E2 -15470.024} C_VEL
LIN {X 0,Y 423.604,Z 383.808,A -85,B 0,C 180,E1 -15470.626,E2 -15470.626} C_VEL
LIN {X 0,Y 419.601,Z 381.497,A -85,B 0,C 180,E1 -15474.667,E2 -15474.667} C_VEL
LIN {X 0,Y 417.71,Z 378.085,A -85,B 0,C 180,E1 -15479.451,E2 -15479.451} C_VEL
LIN {X 0,Y 417.634,Z 377.717,A -85,B 0,C 180,E1 -15480.96,E2 -15480.96} C_VEL
LIN {X 0,Y 417.839,Z 378.527,A -85,B 0,C 180,E1 -15483.018,E2 -15483.018} C_VEL
LIN {X 0,Y 422.288,Z 383.391,A -85,B 0,C 180,E1 -15489.954,E2 -15489.954} C_VEL
LIN {X 0,Y 423.813,Z 384.126,A -85,B 0,C 180,E1 -15491.224,E2 -15491.224} C_VEL
LIN {X 0,Y 425.701,Z 387.832,A -85,B 0,C 180,E1 -15492.824,E2 -15492.824} C_VEL
LIN {X 0,Y 429.146,Z 390.329,A -85,B 0,C 180,E1 -15494.989,E2 -15494.989} C_VEL
LIN {X 0,Y 429.818,Z 390.941,A -85,B 0,C 180,E1 -15495.379,E2 -15495.379} C_VEL
LIN {X 0,Y 432.013,Z 394.604,A -85,B 0,C 180,E1 -15496.678,E2 -15496.678} C_VEL
LIN {X 0,Y 435.424,Z 397.4,A -85,B 0,C 180,E1 -15498.337,E2 -15498.337} C_VEL
LIN {X 0,Y 438.244,Z 401.378,A -85,B 0,C 180,E1 -15499.666,E2 -15499.666} C_VEL
LIN {X 0,Y 440.955,Z 403.845,A -85,B 0,C 180,E1 -15500.786,E2 -15500.786} C_VEL
LIN {X 0,Y 444.176,Z 408.061,A -85,B 0,C 180,E1 -15502.082,E2 -15502.082} C_VEL
LIN {X 0,Y 446.477,Z 410.615,A -85,B 0,C 180,E1 -15502.934,E2 -15502.934} C_VEL
LIN {X 0,Y 453.195,Z 419.578,A -85,B 0,C 180,E1 -15505.272,E2 -15505.272} C_VEL
LIN {X 0,Y 460.636,Z 429.689,A -85,B 0,C 180,E1 -15507.574,E2 -15507.574} C_VEL
LIN {X 0,Y 470.755,Z 444.426,A -85,B 0,C 180,E1 -15510.366,E2 -15510.366} C_VEL
LIN {X 0,Y 479.537,Z 458.096,A -85,B 0,C 180,E1 -15512.545,E2 -15512.545} C_VEL
LIN {X 0,Y 489.467,Z 474.407,A -85,B 0,C 180,E1 -15514.794,E2 -15514.794} C_VEL
LIN {X 0,Y 496.702,Z 487.427,A -85,B 0,C 180,E1 -15516.327,E2 -15516.327} C_VEL
LIN {X 0,Y 483.728,Z 735.625,A -85,B 0,C 180,E1 -15520.202,E2 -15520.202} C_VEL
LIN {X 0,Y 481.602,Z 768.729,A -85,B 0,C 180,E1 -15520.769,E2 -15520.769} C_VEL
LIN {X 0,Y 479.13,Z 790.719,A -85,B 0,C 180,E1 -15521.281,E2 -15521.281} C_VEL
LIN {X 0,Y 475.807,Z 813.833,A -85,B 0,C 180,E1 -15521.979,E2 -15521.979} C_VEL
LIN {X 0,Y 471.826,Z 835.8,A -85,B 0,C 180,E1 -15522.841,E2 -15522.841} C_VEL
LIN {X 0,Y 467.638,Z 856.114,A -85,B 0,C 180,E1 -15523.811,E2 -15523.811} C_VEL
LIN {X 0,Y 461.99,Z 880.16,A -85,B 0,C 180,E1 -15525.212,E2 -15525.212} C_VEL
LIN {X 0,Y 457.262,Z 898.187,A -85,B 0,C 180,E1 -15526.464,E2 -15526.464} C_VEL
LIN {X 0,Y 451.36,Z 919.266,A -85,B 0,C 180,E1 -15528.179,E2 -15528.179} C_VEL
LIN {X 0,Y 445.618,Z 938.045,A -85,B 0,C 180,E1 -15529.995,E2 -15529.995} C_VEL
LIN {X 0,Y 439.979,Z 955.878,A -85,B 0,C 180,E1 -15531.985,E2 -15531.985} C_VEL
LIN {X 0,Y 434.03,Z 973.857,A -85,B 0,C 180,E1 -15534.349,E2 -15534.349} C_VEL
LIN {X 0,Y 429.059,Z 988.884,A -85,B 0,C 180,E1 -15536.634,E2 -15536.634} C_VEL
LIN {X 0,Y 423.726,Z 1005.06,A -85,B 0,C 180,E1 -15539.513,E2 -15539.513} C_VEL
LIN {X 0,Y 419.754,Z 1017.529,A -85,B 0,C 180,E1 -15542.099,E2 -15542.099} C_VEL
LIN {X 0,Y 415.689,Z 1031.121,A -85,B 0,C 180,E1 -15545.409,E2 -15545.409} C_VEL
LIN {X 0,Y 413.024,Z 1040.998,A -85,B 0,C 180,E1 -15548.26,E2 -15548.26} C_VEL
LIN {X 0,Y 410.69,Z 1051.069,A -85,B 0,C 180,E1 -15551.718,E2 -15551.718} C_VEL
LIN {X 0,Y 409.32,Z 1058.297,A -85,B 0,C 180,E1 -15554.778,E2 -15554.778} C_VEL
LIN {X 0,Y 408.442,Z 1064.74,A -85,B 0,C 180,E1 -15558.133,E2 -15558.133} C_VEL
LIN {X 0,Y 408.054,Z 1069.291,A -85,B 0,C 180,E1 -15561.404,E2 -15561.404} C_VEL
LIN {X 0,Y 407.954,Z 1072.088,A -85,B 0,C 180,E1 -15564.233,E2 -15564.233} C_VEL
LIN {X 0,Y 407.947,Z 1073.995,A -85,B 0,C 180,E1 -15567.471,E2 -15567.471} C_VEL
LIN {X 0,Y 407.955,Z 1074.264,A -85,B 0,C 180,E1 -15570.702,E2 -15570.702} C_VEL
LIN {X 0,Y 407.951,Z 1073.433,A -85,B 0,C 180,E1 -15573.372,E2 -15573.372} C_VEL
LIN {X 0,Y 407.96,Z 1071.487,A -85,B 0,C 180,E1 -15576.191,E2 -15576.191} C_VEL
LIN {X 0,Y 408.143,Z 1067.433,A -85,B 0,C 180,E1 -15579.732,E2 -15579.732} C_VEL
LIN {X 0,Y 408.595,Z 1062.575,A -85,B 0,C 180,E1 -15582.723,E2 -15582.723} C_VEL
LIN {X 0,Y 409.573,Z 1055.82,A -85,B 0,C 180,E1 -15586.014,E2 -15586.014} C_VEL
LIN {X 0,Y 411.2,Z 1047.177,A -85,B 0,C 180,E1 -15589.311,E2 -15589.311} C_VEL
LIN {X 0,Y 413.496,Z 1037.346,A -85,B 0,C 180,E1 -15592.462,E2 -15592.462} C_VEL
LIN {X 0,Y 416.616,Z 1025.549,A -85,B 0,C 180,E1 -15595.595,E2 -15595.595} C_VEL
LIN {X 0,Y 420.015,Z 1013.809,A -85,B 0,C 180,E1 -15598.277,E2 -15598.277} C_VEL
LIN {X 0,Y 424.726,Z 998.353,A -85,B 0,C 180,E1 -15601.287,E2 -15601.287} C_VEL
LIN {X 0,Y 429.195,Z 984.073,A -85,B 0,C 180,E1 -15603.674,E2 -15603.674} C_VEL
LIN {X 0,Y 435.115,Z 965.265,A -85,B 0,C 180,E1 -15606.362,E2 -15606.362} C_VEL
LIN {X 0,Y 440.085,Z 949.144,A -85,B 0,C 180,E1 -15608.336,E2 -15608.336} C_VEL
LIN {X 0,Y 445.983,Z 929.298,A -85,B 0,C 180,E1 -15610.429,E2 -15610.429} C_VEL
LIN {X 0,Y 451.189,Z 910.693,A -85,B 0,C 180,E1 -15612.096,E2 -15612.096} C_VEL
LIN {X 0,Y 456.866,Z 889.058,A -85,B 0,C 180,E1 -15613.756,E2 -15613.756} C_VEL
LIN {X 0,Y 461.923,Z 867.619,A -85,B 0,C 180,E1 -15615.116,E2 -15615.116} C_VEL
LIN {X 0,Y 466.68,Z 845.234,A -85,B 0,C 180,E1 -15616.312,E2 -15616.312} C_VEL
LIN {X 0,Y 470.806,Z 822.209,A -85,B 0,C 180,E1 -15617.293,E2 -15617.293} C_VEL
LIN {X 0,Y 474.446,Z 798.599,A -85,B 0,C 180,E1 -15618.097,E2 -15618.097} C_VEL
LIN {X 0,Y 477.272,Z 774.156,A -85,B 0,C 180,E1 -15618.71,E2 -15618.71} C_VEL
LIN {X 0,Y 479.108,Z 750.268,A -85,B 0,C 180,E1 -15619.162,E2 -15619.162} C_VEL
LIN {X 0,Y 491.484,Z 500.014,A -85,B 0,C 180,E1 -15623.073,E2 -15623.073} C_VEL
LIN {X 0,Y 492.133,Z 484.433,A -85,B 0,C 180,E1 -15623.339,E2 -15623.339} C_VEL
LIN {X 0,Y 481.223,Z 465.091,A -85,B 0,C 180,E1 -15625.532,E2 -15625.532} C_VEL
LIN {X 0,Y 471.922,Z 449.921,A -85,B 0,C 180,E1 -15627.549,E2 -15627.549} C_VEL
LIN {X 0,Y 462.572,Z 435.394,A -85,B 0,C 180,E1 -15629.758,E2 -15629.758} C_VEL
LIN {X 0,Y 452.69,Z 421.179,A -85,B 0,C 180,E1 -15632.329,E2 -15632.329} C_VEL
LIN {X 0,Y 444.329,Z 409.768,A -85,B 0,C 180,E1 -15634.758,E2 -15634.758} C_VEL
LIN {X 0,Y 438.133,Z 401.889,A -85,B 0,C 180,E1 -15636.746,E2 -15636.746} C_VEL
LIN {X 0,Y 434.632,Z 398.042,A -85,B 0,C 180,E1 -15637.941,E2 -15637.941} C_VEL
LIN {X 0,Y 433.205,Z 396.022,A -85,B 0,C 180,E1 -15638.47,E2 -15638.47} C_VEL
LIN {X 0,Y 429.823,Z 392.754,A -85,B 0,C 180,E1 -15639.719,E2 -15639.719} C_VEL
LIN {X 0,Y 427.998,Z 389.885,A -85,B 0,C 180,E1 -15640.483,E2 -15640.483} C_VEL
LIN {X 0,Y 424.721,Z 387.166,A -85,B 0,C 180,E1 -15641.824,E2 -15641.824} C_VEL
LIN {X 0,Y 422.415,Z 383.477,A -85,B 0,C 180,E1 -15642.931,E2 -15642.931} C_VEL
LIN {X 0,Y 418.953,Z 381.085,A -85,B 0,C 180,E1 -15644.567,E2 -15644.567} C_VEL
LIN {X 0,Y 417.166,Z 378.034,A -85,B 0,C 180,E1 -15645.601,E2 -15645.601} C_VEL
LIN {X 0,Y 416.708,Z 376.859,A -85,B 0,C 180,E1 -15645.904,E2 -15645.904} C_VEL
LIN {X 0,Y 413.117,Z 375.015,A -85,B 0,C 180,E1 -15647.986,E2 -15647.986} C_VEL
LIN {X 0,Y 411.261,Z 372.43,A -85,B 0,C 180,E1 -15649.352,E2 -15649.352} C_VEL
LIN {X 0,Y 410.558,Z 370.05,A -85,B 0,C 180,E1 -15650.043,E2 -15650.043} C_VEL
LIN {X 0,Y 410.581,Z 370.069,A -85,B 0,C 180,E1 -15653.849,E2 -15653.849} C_VEL
LIN {X 0,Y 410.588,Z 370.079,A -85,B 0,C 180,E1 -15657.767,E2 -15657.767} C_VEL
LIN {X 0,Y 410.584,Z 370.046,A -85,B 0,C 180,E1 -15661.535,E2 -15661.535} C_VEL
LIN {X 0,Y 410.561,Z 370.05,A -85,B 0,C 180,E1 -15665.31,E2 -15665.31} C_VEL
LIN {X 0,Y 410.552,Z 370.081,A -85,B 0,C 180,E1 -15669.109,E2 -15669.109} C_VEL
LIN {X 0,Y 410.586,Z 370.24,A -85,B 0,C 180,E1 -15672.414,E2 -15672.414} C_VEL
LIN {X 0,Y 411.424,Z 372.836,A -85,B 0,C 180,E1 -15673.206,E2 -15673.206} C_VEL
LIN {X 0,Y 413.977,Z 375.683,A -85,B 0,C 180,E1 -15674.978,E2 -15674.978} C_VEL
LIN {X 0,Y 416.823,Z 377.106,A -85,B 0,C 180,E1 -15676.587,E2 -15676.587} C_VEL
LIN {X 0,Y 418.358,Z 380.281,A -85,B 0,C 180,E1 -15677.526,E2 -15677.526} C_VEL
LIN {X 0,Y 420.981,Z 382.788,A -85,B 0,C 180,E1 -15678.846,E2 -15678.846} C_VEL
LIN {X 0,Y 422.785,Z 383.886,A -85,B 0,C 180,E1 -15679.659,E2 -15679.659} C_VEL
LIN {X 0,Y 424.891,Z 387.415,A -85,B 0,C 180,E1 -15680.671,E2 -15680.671} C_VEL
LIN {X 0,Y 428.425,Z 390.389,A -85,B 0,C 180,E1 -15682.107,E2 -15682.107} C_VEL
LIN {X 0,Y 431.175,Z 394.303,A -85,B 0,C 180,E1 -15683.218,E2 -15683.218} C_VEL
LIN {X 0,Y 433.863,Z 396.716,A -85,B 0,C 180,E1 -15684.183,E2 -15684.183} C_VEL
LIN {X 0,Y 437.263,Z 401.125,A -85,B 0,C 180,E1 -15685.389,E2 -15685.389} C_VEL
LIN {X 0,Y 439.121,Z 403.021,A -85,B 0,C 180,E1 -15685.997,E2 -15685.997} C_VEL
LIN {X 0,Y 442.898,Z 407.603,A -85,B 0,C 180,E1 -15687.205,E2 -15687.205} C_VEL
LIN {X 0,Y 448.961,Z 415.194,A -85,B 0,C 180,E1 -15689.01,E2 -15689.01} C_VEL
LIN {X 0,Y 453.778,Z 421.318,A -85,B 0,C 180,E1 -15690.341,E2 -15690.341} C_VEL
LIN {X 0,Y 461.047,Z 430.651,A -85,B 0,C 180,E1 -15692.206,E2 -15692.206} C_VEL
LIN {X 0,Y 471.423,Z 444.915,A -85,B 0,C 180,E1 -15694.641,E2 -15694.641} C_VEL
LIN {X 0,Y 482.75,Z 461.466,A -85,B 0,C 180,E1 -15697.047,E2 -15697.047} C_VEL
LIN {X 0,Y 492.491,Z 476.892,A -85,B 0,C 180,E1 -15698.956,E2 -15698.956} C_VEL
LIN {X 0,Y 479.792,Z 731.368,A -85,B 0,C 180,E1 -15702.926,E2 -15702.926} C_VEL
LIN {X 0,Y 477.984,Z 756.062,A -85,B 0,C 180,E1 -15703.392,E2 -15703.392} C_VEL
LIN {X 0,Y 475.502,Z 779.25,A -85,B 0,C 180,E1 -15703.985,E2 -15703.985} C_VEL
LIN {X 0,Y 472.191,Z 802.335,A -85,B 0,C 180,E1 -15704.772,E2 -15704.772} C_VEL
LIN {X 0,Y 468.813,Z 822.107,A -85,B 0,C 180,E1 -15705.608,E2 -15705.608} C_VEL
LIN {X 0,Y 464.329,Z 844.943,A -85,B 0,C 180,E1 -15706.781,E2 -15706.781} C_VEL
LIN {X 0,Y 459.73,Z 864.986,A -85,B 0,C 180,E1 -15708.026,E2 -15708.026} C_VEL
LIN {X 0,Y 454.482,Z 886.14,A -85,B 0,C 180,E1 -15709.573,E2 -15709.573} C_VEL
LIN {X 0,Y 449.076,Z 905.598,A -85,B 0,C 180,E1 -15711.269,E2 -15711.269} C_VEL
LIN {X 0,Y 443.95,Z 923.103,A -85,B 0,C 180,E1 -15713.033,E2 -15713.033} C_VEL
LIN {X 0,Y 437.883,Z 942.682,A -85,B 0,C 180,E1 -15715.349,E2 -15715.349} C_VEL
LIN {X 0,Y 432.985,Z 957.931,A -85,B 0,C 180,E1 -15717.448,E2 -15717.448} C_VEL
LIN {X 0,Y 427.321,Z 975.393,A -85,B 0,C 180,E1 -15720.26,E2 -15720.26} C_VEL
LIN {X 0,Y 423.112,Z 988.41,A -85,B 0,C 180,E1 -15722.712,E2 -15722.712} C_VEL
LIN {X 0,Y 418.604,Z 1002.813,A -85,B 0,C 180,E1 -15725.892,E2 -15725.892} C_VEL
LIN {X 0,Y 415.435,Z 1013.514,A -85,B 0,C 180,E1 -15728.689,E2 -15728.689} C_VEL
LIN {X 0,Y 412.531,Z 1024.412,A -85,B 0,C 180,E1 -15732.072,E2 -15732.072} C_VEL
LIN {X 0,Y 410.692,Z 1032.286,A -85,B 0,C 180,E1 -15735.044,E2 -15735.044} C_VEL
LIN {X 0,Y 409.303,Z 1039.625,A -85,B 0,C 180,E1 -15738.411,E2 -15738.411} C_VEL
LIN {X 0,Y 408.523,Z 1044.83,A -85,B 0,C 180,E1 -15741.555,E2 -15741.555} C_VEL
LIN {X 0,Y 408.159,Z 1048.539,A -85,B 0,C 180,E1 -15744.518,E2 -15744.518} C_VEL
LIN {X 0,Y 407.999,Z 1051.38,A -85,B 0,C 180,E1 -15748.034,E2 -15748.034} C_VEL
LIN {X 0,Y 407.964,Z 1052.407,A -85,B 0,C 180,E1 -15750.843,E2 -15750.843} C_VEL
LIN {X 0,Y 407.96,Z 1052.4,A -85,B 0,C 180,E1 -15753.654,E2 -15753.654} C_VEL
LIN {X 0,Y 408.018,Z 1051.383,A -85,B 0,C 180,E1 -15756.417,E2 -15756.417} C_VEL
LIN {X 0,Y 407.067,Z 1050.788,A -85,B 0,C 180,E1 -15757.496,E2 -15757.496} C_VEL
LIN {X 0,Y 400.81,Z 1048.289,A -85,B 0,C 180,E1 -15760.53,E2 -15760.53} C_VEL
LIN {X 0,Y 400.372,Z 1047.462,A -85,B 0,C 180,E1 -15761.318,E2 -15761.318} C_VEL
LIN {X 0,Y 401.121,Z 1042.412,A -85,B 0,C 180,E1 -15764.877,E2 -15764.877} C_VEL
LIN {X 0,Y 402.193,Z 1036.974,A -85,B 0,C 180,E1 -15767.806,E2 -15767.806} C_VEL
LIN {X 0,Y 404.102,Z 1029.272,A -85,B 0,C 180,E1 -15771.177,E2 -15771.177} C_VEL
LIN {X 0,Y 406.684,Z 1020.075,A -85,B 0,C 180,E1 -15774.397,E2 -15774.397} C_VEL
LIN {X 0,Y 410.136,Z 1009.29,A -85,B 0,C 180,E1 -15777.594,E2 -15777.594} C_VEL
LIN {X 0,Y 414.282,Z 997.002,A -85,B 0,C 180,E1 -15780.614,E2 -15780.614} C_VEL
LIN {X 0,Y 418.81,Z 984.227,A -85,B 0,C 180,E1 -15783.32,E2 -15783.32} C_VEL
LIN {X 0,Y 424.332,Z 968.783,A -85,B 0,C 180,E1 -15786.093,E2 -15786.093} C_VEL
LIN {X 0,Y 429.412,Z 954.485,A -85,B 0,C 180,E1 -15788.306,E2 -15788.306} C_VEL
LIN {X 0,Y 435.981,Z 935.537,A -85,B 0,C 180,E1 -15790.816,E2 -15790.816} C_VEL
LIN {X 0,Y 441.536,Z 918.763,A -85,B 0,C 180,E1 -15792.706,E2 -15792.706} C_VEL
LIN {X 0,Y 447.949,Z 898.327,A -85,B 0,C 180,E1 -15794.678,E2 -15794.678} C_VEL
LIN {X 0,Y 453.407,Z 879.276,A -85,B 0,C 180,E1 -15796.231,E2 -15796.231} C_VEL
LIN {X 0,Y 458.932,Z 858.441,A -85,B 0,C 180,E1 -15797.683,E2 -15797.683} C_VEL
LIN {X 0,Y 464.038,Z 836.256,A -85,B 0,C 180,E1 -15798.953,E2 -15798.953} C_VEL
LIN {X 0,Y 468.264,Z 815.417,A -85,B 0,C 180,E1 -15799.952,E2 -15799.952} C_VEL
LIN {X 0,Y 472.296,Z 791.455,A -85,B 0,C 180,E1 -15800.87,E2 -15800.87} C_VEL
LIN {X 0,Y 475.196,Z 770.065,A -85,B 0,C 180,E1 -15801.513,E2 -15801.513} C_VEL
LIN {X 0,Y 477.824,Z 743.477,A -85,B 0,C 180,E1 -15802.099,E2 -15802.099} C_VEL
LIN {X 0,Y 490.209,Z 516.941,A -85,B 0,C 180,E1 -15805.673,E2 -15805.673} C_VEL
LIN {X 0,Y 491.989,Z 483.415,A -85,B 0,C 180,E1 -15806.213,E2 -15806.213} C_VEL
LIN {X 0,Y 480.98,Z 466.388,A -85,B 0,C 180,E1 -15808.617,E2 -15808.617} C_VEL
LIN {X 0,Y 471.213,Z 452.45,A -85,B 0,C 180,E1 -15810.961,E2 -15810.961} C_VEL
LIN {X 0,Y 463.001,Z 441.37,A -85,B 0,C 180,E1 -15813.135,E2 -15813.135} C_VEL
LIN {X 0,Y 455.92,Z 432.167,A -85,B 0,C 180,E1 -15815.201,E2 -15815.201} C_VEL
LIN {X 0,Y 451.75,Z 426.891,A -85,B 0,C 180,E1 -15816.521,E2 -15816.521} C_VEL
LIN {X 0,Y 447.528,Z 421.652,A -85,B 0,C 180,E1 -15817.954,E2 -15817.954} C_VEL
LIN {X 0,Y 443.072,Z 416.189,A -85,B 0,C 180,E1 -15819.594,E2 -15819.594} C_VEL
LIN {X 0,Y 439.439,Z 411.92,A -85,B 0,C 180,E1 -15821.046,E2 -15821.046} C_VEL
LIN {X 0,Y 438.344,Z 410.514,A -85,B 0,C 180,E1 -15821.514,E2 -15821.514} C_VEL
LIN {X 0,Y 434.931,Z 406.953,A -85,B 0,C 180,E1 -15823.024,E2 -15823.024} C_VEL
LIN {X 0,Y 433.411,Z 404.566,A -85,B 0,C 180,E1 -15823.79,E2 -15823.79} C_VEL
LIN {X 0,Y 429.882,Z 401.428,A -85,B 0,C 180,E1 -15825.589,E2 -15825.589} C_VEL
LIN {X 0,Y 427.982,Z 398.219,A -85,B 0,C 180,E1 -15826.764,E2 -15826.764} C_VEL
LIN {X 0,Y 424.655,Z 395.833,A -85,B 0,C 180,E1 -15828.868,E2 -15828.868} C_VEL
LIN {X 0,Y 422.725,Z 392.54,A -85,B 0,C 180,E1 -15830.469,E2 -15830.469} C_VEL
LIN {X 0,Y 422.299,Z 391.674,A -85,B 0,C 180,E1 -15830.872,E2 -15830.872} C_VEL
LIN {X 0,Y 418.26,Z 389.093,A -85,B 0,C 180,E1 -15835.2,E2 -15835.2} C_VEL
LIN {X 0,Y 416.718,Z 385.975,A -85,B 0,C 180,E1 -15839.588,E2 -15839.588} C_VEL
LIN {X 0,Y 416.659,Z 385.66,A -85,B 0,C 180,E1 -15840.963,E2 -15840.963} C_VEL
LIN {X 0,Y 416.861,Z 386.506,A -85,B 0,C 180,E1 -15843.025,E2 -15843.025} C_VEL
LIN {X 0,Y 421.336,Z 391.347,A -85,B 0,C 180,E1 -15849.985,E2 -15849.985} C_VEL
LIN {X 0,Y 422.519,Z 391.901,A -85,B 0,C 180,E1 -15850.982,E2 -15850.982} C_VEL
LIN {X 0,Y 424.546,Z 395.749,A -85,B 0,C 180,E1 -15852.722,E2 -15852.722} C_VEL
LIN {X 0,Y 428.342,Z 398.664,A -85,B 0,C 180,E1 -15855.121,E2 -15855.121} C_VEL
LIN {X 0,Y 430.683,Z 402.432,A -85,B 0,C 180,E1 -15856.523,E2 -15856.523} C_VEL
LIN {X 0,Y 433.847,Z 405.141,A -85,B 0,C 180,E1 -15858.093,E2 -15858.093} C_VEL
LIN {X 0,Y 436.854,Z 409.216,A -85,B 0,C 180,E1 -15859.522,E2 -15859.522} C_VEL
LIN {X 0,Y 439.157,Z 411.365,A -85,B 0,C 180,E1 -15860.491,E2 -15860.491} C_VEL
LIN {X 0,Y 442.576,Z 415.762,A -85,B 0,C 180,E1 -15861.887,E2 -15861.887} C_VEL
LIN {X 0,Y 444.917,Z 418.595,A -85,B 0,C 180,E1 -15862.775,E2 -15862.775} C_VEL
LIN {X 0,Y 450.958,Z 426.734,A -85,B 0,C 180,E1 -15864.915,E2 -15864.915} C_VEL
LIN {X 0,Y 458.382,Z 436.992,A -85,B 0,C 180,E1 -15867.264,E2 -15867.264} C_VEL
LIN {X 0,Y 468.267,Z 451.648,A -85,B 0,C 180,E1 -15870.048,E2 -15870.048} C_VEL
LIN {X 0,Y 478.528,Z 467.841,A -85,B 0,C 180,E1 -15872.622,E2 -15872.622} C_VEL
LIN {X 0,Y 489.337,Z 486.411,A -85,B 0,C 180,E1 -15875.078,E2 -15875.078} C_VEL
LIN {X 0,Y 491.861,Z 491.262,A -85,B 0,C 180,E1 -15875.628,E2 -15875.628} C_VEL
LIN {X 0,Y 478.418,Z 740.475,A -85,B 0,C 180,E1 -15879.538,E2 -15879.538} C_VEL
LIN {X 0,Y 476.271,Z 770.622,A -85,B 0,C 180,E1 -15880.072,E2 -15880.072} C_VEL
LIN {X 0,Y 473.736,Z 792.208,A -85,B 0,C 180,E1 -15880.585,E2 -15880.585} C_VEL
LIN {X 0,Y 469.904,Z 817.136,A -85,B 0,C 180,E1 -15881.368,E2 -15881.368} C_VEL
LIN {X 0,Y 466.109,Z 837.319,A -85,B 0,C 180,E1 -15882.179,E2 -15882.179} C_VEL
LIN {X 0,Y 461.364,Z 859.57,A -85,B 0,C 180,E1 -15883.265,E2 -15883.265} C_VEL
LIN {X 0,Y 456.01,Z 881.169,A -85,B 0,C 180,E1 -15884.561,E2 -15884.561} C_VEL
LIN {X 0,Y 450.954,Z 899.799,A -85,B 0,C 180,E1 -15885.875,E2 -15885.875} C_VEL
LIN {X 0,Y 444.342,Z 922.247,A -85,B 0,C 180,E1 -15887.761,E2 -15887.761} C_VEL
LIN {X 0,Y 438.975,Z 939.213,A -85,B 0,C 180,E1 -15889.437,E2 -15889.437} C_VEL
LIN {X 0,Y 432.809,Z 957.929,A -85,B 0,C 180,E1 -15891.578,E2 -15891.578} C_VEL
LIN {X 0,Y 427.03,Z 974.683,A -85,B 0,C 180,E1 -15893.839,E2 -15893.839} C_VEL
LIN {X 0,Y 421.34,Z 991.304,A -85,B 0,C 180,E1 -15896.431,E2 -15896.431} C_VEL
LIN {X 0,Y 416.125,Z 1006.337,A -85,B 0,C 180,E1 -15899.216,E2 -15899.216} C_VEL
LIN {X 0,Y 411.569,Z 1020.223,A -85,B 0,C 180,E1 -15902.196,E2 -15902.196} C_VEL
LIN {X 0,Y 407.702,Z 1032.524,A -85,B 0,C 180,E1 -15905.359,E2 -15905.359} C_VEL
LIN {X 0,Y 404.684,Z 1043.503,A -85,B 0,C 180,E1 -15908.669,E2 -15908.669} C_VEL
LIN {X 0,Y 402.573,Z 1052.271,A -85,B 0,C 180,E1 -15911.913,E2 -15911.913} C_VEL
LIN {X 0,Y 401.249,Z 1059.188,A -85,B 0,C 180,E1 -15914.98,E2 -15914.98} C_VEL
LIN {X 0,Y 400.357,Z 1065.613,A -85,B 0,C 180,E1 -15918.621,E2 -15918.621} C_VEL
LIN {X 0,Y 400.047,Z 1069.421,A -85,B 0,C 180,E1 -15921.52,E2 -15921.52} C_VEL
LIN {X 0,Y 399.951,Z 1072.235,A -85,B 0,C 180,E1 -15924.549,E2 -15924.549} C_VEL
LIN {X 0,Y 399.951,Z 1073.892,A -85,B 0,C 180,E1 -15927.994,E2 -15927.994} C_VEL
LIN {X 0,Y 399.959,Z 1074.025,A -85,B 0,C 180,E1 -15930.859,E2 -15930.859} C_VEL
LIN {X 0,Y 399.948,Z 1073.142,A -85,B 0,C 180,E1 -15933.583,E2 -15933.583} C_VEL
LIN {X 0,Y 399.964,Z 1070.909,A -85,B 0,C 180,E1 -15936.748,E2 -15936.748} C_VEL
LIN {X 0,Y 400.185,Z 1066.77,A -85,B 0,C 180,E1 -15940.218,E2 -15940.218} C_VEL
LIN {X 0,Y 400.678,Z 1062.068,A -85,B 0,C 180,E1 -15943.126,E2 -15943.126} C_VEL
LIN {X 0,Y 401.756,Z 1055.217,A -85,B 0,C 180,E1 -15946.482,E2 -15946.482} C_VEL
LIN {X 0,Y 403.429,Z 1046.909,A -85,B 0,C 180,E1 -15949.699,E2 -15949.699} C_VEL
LIN {X 0,Y 405.86,Z 1037.07,A -85,B 0,C 180,E1 -15952.908,E2 -15952.908} C_VEL
LIN {X 0,Y 409.143,Z 1025.257,A -85,B 0,C 180,E1 -15956.097,E2 -15956.097} C_VEL
LIN {X 0,Y 412.928,Z 1012.863,A -85,B 0,C 180,E1 -15958.966,E2 -15958.966} C_VEL
LIN {X 0,Y 417.745,Z 997.718,A -85,B 0,C 180,E1 -15961.936,E2 -15961.936} C_VEL
LIN {X 0,Y 422.315,Z 983.746,A -85,B 0,C 180,E1 -15964.298,E2 -15964.298} C_VEL
LIN {X 0,Y 428.308,Z 965.43,A -85,B 0,C 180,E1 -15966.951,E2 -15966.951} C_VEL
LIN {X 0,Y 433.27,Z 949.908,A -85,B 0,C 180,E1 -15968.882,E2 -15968.882} C_VEL
LIN {X 0,Y 439.257,Z 930.606,A -85,B 0,C 180,E1 -15970.964,E2 -15970.964} C_VEL
LIN {X 0,Y 444.915,Z 911.03,A -85,B 0,C 180,E1 -15972.743,E2 -15972.743} C_VEL
LIN {X 0,Y 450.545,Z 890.396,A -85,B 0,C 180,E1 -15974.353,E2 -15974.353} C_VEL
LIN {X 0,Y 455.813,Z 868.823,A -85,B 0,C 180,E1 -15975.744,E2 -15975.744} C_VEL
LIN {X 0,Y 460.577,Z 847.137,A -85,B 0,C 180,E1 -15976.922,E2 -15976.922} C_VEL
LIN {X 0,Y 464.961,Z 823.854,A -85,B 0,C 180,E1 -15977.941,E2 -15977.941} C_VEL
LIN {X 0,Y 468.475,Z 801.857,A -85,B 0,C 180,E1 -15978.709,E2 -15978.709} C_VEL
LIN {X 0,Y 471.729,Z 775.805,A -85,B 0,C 180,E1 -15979.392,E2 -15979.392} C_VEL
LIN {X 0,Y 473.577,Z 753.395,A -85,B 0,C 180,E1 -15979.828,E2 -15979.828} C_VEL
LIN {X 0,Y 486.271,Z 505.898,A -85,B 0,C 180,E1 -15983.725,E2 -15983.725} C_VEL
LIN {X 0,Y 487.071,Z 488.034,A -85,B 0,C 180,E1 -15984.028,E2 -15984.028} C_VEL
LIN {X 0,Y 476.42,Z 469.074,A -85,B 0,C 180,E1 -15986.245,E2 -15986.245} C_VEL
LIN {X 0,Y 465.987,Z 451.929,A -85,B 0,C 180,E1 -15988.609,E2 -15988.609} C_VEL
LIN {X 0,Y 455.615,Z 436.082,A -85,B 0,C 180,E1 -15991.202,E2 -15991.202} C_VEL
LIN {X 0,Y 448.887,Z 426.559,A -85,B 0,C 180,E1 -15993.045,E2 -15993.045} C_VEL
LIN {X 0,Y 441.99,Z 416.9,A -85,B 0,C 180,E1 -15995.116,E2 -15995.116} C_VEL
LIN {X 0,Y 435.88,Z 409.12,A -85,B 0,C 180,E1 -15997.118,E2 -15997.118} C_VEL
LIN {X 0,Y 432.286,Z 404.919,A -85,B 0,C 180,E1 -15998.386,E2 -15998.386} C_VEL
LIN {X 0,Y 431.029,Z 403.342,A -85,B 0,C 180,E1 -15998.855,E2 -15998.855} C_VEL
LIN {X 0,Y 427.579,Z 399.663,A -85,B 0,C 180,E1 -16000.179,E2 -16000.179} C_VEL
LIN {X 0,Y 426.075,Z 397.406,A -85,B 0,C 180,E1 -16000.819,E2 -16000.819} C_VEL
LIN {X 0,Y 422.735,Z 394.337,A -85,B 0,C 180,E1 -16002.234,E2 -16002.234} C_VEL
LIN {X 0,Y 420.881,Z 391.233,A -85,B 0,C 180,E1 -16003.152,E2 -16003.152} C_VEL
LIN {X 0,Y 417.351,Z 388.627,A -85,B 0,C 180,E1 -16004.862,E2 -16004.862} C_VEL
LIN {X 0,Y 415.389,Z 385.174,A -85,B 0,C 180,E1 -16006.036,E2 -16006.036} C_VEL
LIN {X 0,Y 414.878,Z 384.579,A -85,B 0,C 180,E1 -16006.338,E2 -16006.338} C_VEL
LIN {X 0,Y 411.246,Z 382.217,A -85,B 0,C 180,E1 -16008.571,E2 -16008.571} C_VEL
LIN {X 0,Y 409.506,Z 379.103,A -85,B 0,C 180,E1 -16009.981,E2 -16009.981} C_VEL
LIN {X 0,Y 409.032,Z 377.905,A -85,B 0,C 180,E1 -16010.431,E2 -16010.431} C_VEL
LIN {X 0,Y 405.105,Z 375.919,A -85,B 0,C 180,E1 -16014.192,E2 -16014.192} C_VEL
LIN {X 0,Y 402.692,Z 371.474,A -85,B 0,C 180,E1 -16020.142,E2 -16020.142} C_VEL
LIN {X 0,Y 402.678,Z 371.328,A -85,B 0,C 180,E1 -16021.992,E2 -16021.992} C_VEL
LIN {X 0,Y 403.829,Z 374.366,A -85,B 0,C 180,E1 -16026.255,E2 -16026.255} C_VEL
LIN {X 0,Y 407.511,Z 377.451,A -85,B 0,C 180,E1 -16030.747,E2 -16030.747} C_VEL
LIN {X 0,Y 409.198,Z 378.17,A -85,B 0,C 180,E1 -16032.131,E2 -16032.131} C_VEL
LIN {X 0,Y 410.435,Z 381.109,A -85,B 0,C 180,E1 -16033.238,E2 -16033.238} C_VEL
LIN {X 0,Y 413.249,Z 383.839,A -85,B 0,C 180,E1 -16035.148,E2 -16035.148} C_VEL
LIN {X 0,Y 415.252,Z 384.872,A -85,B 0,C 180,E1 -16036.291,E2 -16036.291} C_VEL
LIN {X 0,Y 417.204,Z 388.397,A -85,B 0,C 180,E1 -16037.472,E2 -16037.472} C_VEL
LIN {X 0,Y 420.046,Z 390.833,A -85,B 0,C 180,E1 -16038.889,E2 -16038.889} C_VEL
LIN {X 0,Y 421.105,Z 391.631,A -85,B 0,C 180,E1 -16039.38,E2 -16039.38} C_VEL
LIN {X 0,Y 423.636,Z 395.448,A -85,B 0,C 180,E1 -16040.59,E2 -16040.59} C_VEL
LIN {X 0,Y 426.588,Z 397.977,A -85,B 0,C 180,E1 -16041.809,E2 -16041.809} C_VEL
LIN {X 0,Y 429.558,Z 402.02,A -85,B 0,C 180,E1 -16043.02,E2 -16043.02} C_VEL
LIN {X 0,Y 431.947,Z 404.299,A -85,B 0,C 180,E1 -16043.897,E2 -16043.897} C_VEL
LIN {X 0,Y 435.591,Z 408.847,A -85,B 0,C 180,E1 -16045.202,E2 -16045.202} C_VEL
LIN {X 0,Y 437.227,Z 410.734,A -85,B 0,C 180,E1 -16045.754,E2 -16045.754} C_VEL
LIN {X 0,Y 442.213,Z 416.886,A -85,B 0,C 180,E1 -16047.36,E2 -16047.36} C_VEL
LIN {X 0,Y 446.77,Z 422.643,A -85,B 0,C 180,E1 -16048.726,E2 -16048.726} C_VEL
LIN {X 0,Y 451.748,Z 429.041,A -85,B 0,C 180,E1 -16050.125,E2 -16050.125} C_VEL
LIN {X 0,Y 458.95,Z 438.496,A -85,B 0,C 180,E1 -16052.003,E2 -16052.003} C_VEL
LIN {X 0,Y 468.414,Z 451.673,A -85,B 0,C 180,E1 -16054.264,E2 -16054.264} C_VEL
LIN {X 0,Y 479.358,Z 467.882,A -85,B 0,C 180,E1 -16056.643,E2 -16056.643} C_VEL
LIN {X 0,Y 487.422,Z 480.855,A -85,B 0,C 180,E1 -16058.272,E2 -16058.272} C_VEL
LIN {X 0,Y 474.319,Z 734.433,A -85,B 0,C 180,E1 -16062.254,E2 -16062.254} C_VEL
LIN {X 0,Y 472.532,Z 757.416,A -85,B 0,C 180,E1 -16062.699,E2 -16062.699} C_VEL
LIN {X 0,Y 469.826,Z 781.616,A -85,B 0,C 180,E1 -16063.333,E2 -16063.333} C_VEL
LIN {X 0,Y 466.49,Z 803.749,A -85,B 0,C 180,E1 -16064.106,E2 -16064.106} C_VEL
LIN {X 0,Y 462.682,Z 825.268,A -85,B 0,C 180,E1 -16065.035,E2 -16065.035} C_VEL
LIN {X 0,Y 457.838,Z 848.459,A -85,B 0,C 180,E1 -16066.274,E2 -16066.274} C_VEL
LIN {X 0,Y 453.361,Z 867.266,A -85,B 0,C 180,E1 -16067.469,E2 -16067.469} C_VEL
LIN {X 0,Y 447.651,Z 889.182,A -85,B 0,C 180,E1 -16069.122,E2 -16069.122} C_VEL
LIN {X 0,Y 442.417,Z 907.348,A -85,B 0,C 180,E1 -16070.742,E2 -16070.742} C_VEL
LIN {X 0,Y 436.621,Z 926.505,A -85,B 0,C 180,E1 -16072.719,E2 -16072.719} C_VEL
LIN {X 0,Y 430.734,Z 944.563,A -85,B 0,C 180,E1 -16074.933,E2 -16074.933} C_VEL
LIN {X 0,Y 425.023,Z 961.78,A -85,B 0,C 180,E1 -16077.375,E2 -16077.375} C_VEL
LIN {X 0,Y 419.749,Z 977.254,A -85,B 0,C 180,E1 -16079.984,E2 -16079.984} C_VEL
LIN {X 0,Y 415.005,Z 991.499,A -85,B 0,C 180,E1 -16082.756,E2 -16082.756} C_VEL
LIN {X 0,Y 410.81,Z 1004.252,A -85,B 0,C 180,E1 -16085.711,E2 -16085.711} C_VEL
LIN {X 0,Y 407.422,Z 1015.332,A -85,B 0,C 180,E1 -16088.702,E2 -16088.702} C_VEL
LIN {X 0,Y 404.585,Z 1025.491,A -85,B 0,C 180,E1 -16092.006,E2 -16092.006} C_VEL
LIN {X 0,Y 402.711,Z 1033.254,A -85,B 0,C 180,E1 -16095.036,E2 -16095.036} C_VEL
LIN {X 0,Y 401.241,Z 1040.688,A -85,B 0,C 180,E1 -16098.646,E2 -16098.646} C_VEL
LIN {X 0,Y 400.515,Z 1045.483,A -85,B 0,C 180,E1 -16101.674,E2 -16101.674} C_VEL
LIN {X 0,Y 400.13,Z 1049.406,A -85,B 0,C 180,E1 -16104.982,E2 -16104.982} C_VEL
LIN {X 0,Y 399.993,Z 1051.738,A -85,B 0,C 180,E1 -16108.281,E2 -16108.281} C_VEL
LIN {X 0,Y 399.963,Z 1052.647,A -85,B 0,C 180,E1 -16111.003,E2 -16111.003} C_VEL
LIN {X 0,Y 399.966,Z 1052.589,A -85,B 0,C 180,E1 -16113.87,E2 -16113.87} C_VEL
LIN {X 0,Y 400.05,Z 1051.129,A -85,B 0,C 180,E1 -16117.323,E2 -16117.323} C_VEL
LIN {X 0,Y 400.254,Z 1048.492,A -85,B 0,C 180,E1 -16120.362,E2 -16120.362} C_VEL
LIN {X 0,Y 400.372,Z 1047.462,A -85,B 0,C 180,E1 -16121.318,E2 -16121.318} C_VEL
LIN {X 0,Y 399.552,Z 1046.226,A -85,B 0,C 180,E1 -16122.409,E2 -16122.409} C_VEL
LIN {X 0,Y 393.933,Z 1042.172,A -85,B 0,C 180,E1 -16125.401,E2 -16125.401} C_VEL
LIN {X 0,Y 393.592,Z 1040.769,A -85,B 0,C 180,E1 -16126.269,E2 -16126.269} C_VEL
LIN {X 0,Y 395.335,Z 1033.293,A -85,B 0,C 180,E1 -16129.965,E2 -16129.965} C_VEL
LIN {X 0,Y 397.439,Z 1025.806,A -85,B 0,C 180,E1 -16132.957,E2 -16132.957} C_VEL
LIN {X 0,Y 400.862,Z 1015.037,A -85,B 0,C 180,E1 -16136.519,E2 -16136.519} C_VEL
LIN {X 0,Y 404.547,Z 1004.329,A -85,B 0,C 180,E1 -16139.463,E2 -16139.463} C_VEL
LIN {X 0,Y 409.456,Z 990.937,A -85,B 0,C 180,E1 -16142.596,E2 -16142.596} C_VEL
LIN {X 0,Y 414.371,Z 977.647,A -85,B 0,C 180,E1 -16145.22,E2 -16145.22} C_VEL
LIN {X 0,Y 420.216,Z 962.118,A -85,B 0,C 180,E1 -16147.872,E2 -16147.872} C_VEL
LIN {X 0,Y 426.245,Z 945.497,A -85,B 0,C 180,E1 -16150.261,E2 -16150.261} C_VEL
LIN {X 0,Y 432.123,Z 928.921,A -85,B 0,C 180,E1 -16152.326,E2 -16152.326} C_VEL
LIN {X 0,Y 438.674,Z 909.227,A -85,B 0,C 180,E1 -16154.408,E2 -16154.408} C_VEL
LIN {X 0,Y 444.103,Z 891.864,A -85,B 0,C 180,E1 -16155.978,E2 -16155.978} C_VEL
LIN {X 0,Y 450.388,Z 869.901,A -85,B 0,C 180,E1 -16157.67,E2 -16157.67} C_VEL
LIN {X 0,Y 455.489,Z 850.06,A -85,B 0,C 180,E1 -16158.943,E2 -16158.943} C_VEL
LIN {X 0,Y 460.518,Z 828.114,A -85,B 0,C 180,E1 -16160.133,E2 -16160.133} C_VEL
LIN {X 0,Y 464.9,Z 805.136,A -85,B 0,C 180,E1 -16161.13,E2 -16161.13} C_VEL
LIN {X 0,Y 468.531,Z 782.725,A -85,B 0,C 180,E1 -16161.913,E2 -16161.913} C_VEL
LIN {X 0,Y 471.493,Z 758.274,A -85,B 0,C 180,E1 -16162.555,E2 -16162.555} C_VEL
LIN {X 0,Y 473.398,Z 735.671,A -85,B 0,C 180,E1 -16162.993,E2 -16162.993} C_VEL
LIN {X 0,Y 487.324,Z 487.631,A -85,B 0,C 180,E1 -16166.904,E2 -16166.904} C_VEL
LIN {X 0,Y 476.642,Z 471.149,A -85,B 0,C 180,E1 -16169.317,E2 -16169.317} C_VEL
LIN {X 0,Y 468.164,Z 458.897,A -85,B 0,C 180,E1 -16171.418,E2 -16171.418} C_VEL
LIN {X 0,Y 460.095,Z 447.835,A -85,B 0,C 180,E1 -16173.613,E2 -16173.613} C_VEL
LIN {X 0,Y 453.331,Z 438.974,A -85,B 0,C 180,E1 -16175.641,E2 -16175.641} C_VEL
LIN {X 0,Y 449.328,Z 433.847,A -85,B 0,C 180,E1 -16176.942,E2 -16176.942} C_VEL
LIN {X 0,Y 445.527,Z 429.019,A -85,B 0,C 180,E1 -16178.265,E2 -16178.265} C_VEL
LIN {X 0,Y 441.138,Z 423.591,A -85,B 0,C 180,E1 -16179.916,E2 -16179.916} C_VEL
LIN {X 0,Y 437.433,Z 419.055,A -85,B 0,C 180,E1 -16181.44,E2 -16181.44} C_VEL
LIN {X 0,Y 432.902,Z 413.914,A -85,B 0,C 180,E1 -16183.495,E2 -16183.495} C_VEL
LIN {X 0,Y 431.916,Z 412.287,A -85,B 0,C 180,E1 -16184.009,E2 -16184.009} C_VEL
LIN {X 0,Y 428.332,Z 408.967,A -85,B 0,C 180,E1 -16185.881,E2 -16185.881} C_VEL
LIN {X 0,Y 426.568,Z 406.004,A -85,B 0,C 180,E1 -16186.995,E2 -16186.995} C_VEL
LIN {X 0,Y 423.227,Z 403.422,A -85,B 0,C 180,E1 -16189.174,E2 -16189.174} C_VEL
LIN {X 0,Y 421.302,Z 399.897,A -85,B 0,C 180,E1 -16190.85,E2 -16190.85} C_VEL
LIN {X 0,Y 416.05,Z 394.962,A -85,B 0,C 180,E1 -16197.934,E2 -16197.934} C_VEL
LIN {X 0,Y 415.69,Z 393.552,A -85,B 0,C 180,E1 -16200.689,E2 -16200.689} C_VEL
LIN {X 0,Y 415.834,Z 394.29,A -85,B 0,C 180,E1 -16202.756,E2 -16202.756} C_VEL
LIN {X 0,Y 420.213,Z 399.241,A -85,B 0,C 180,E1 -16209.865,E2 -16209.865} C_VEL
LIN {X 0,Y 421.299,Z 399.833,A -85,B 0,C 180,E1 -16210.807,E2 -16210.807} C_VEL
LIN {X 0,Y 423.392,Z 403.66,A -85,B 0,C 180,E1 -16212.618,E2 -16212.618} C_VEL
LIN {X 0,Y 426.925,Z 406.472,A -85,B 0,C 180,E1 -16214.895,E2 -16214.895} C_VEL
LIN {X 0,Y 429.477,Z 410.381,A -85,B 0,C 180,E1 -16216.432,E2 -16216.432} C_VEL
LIN {X 0,Y 432.221,Z 412.744,A -85,B 0,C 180,E1 -16217.815,E2 -16217.815} C_VEL
LIN {X 0,Y 435.466,Z 417.05,A -85,B 0,C 180,E1 -16219.378,E2 -16219.378} C_VEL
LIN {X 0,Y 437.511,Z 419.106,A -85,B 0,C 180,E1 -16220.258,E2 -16220.258} C_VEL
LIN {X 0,Y 441.143,Z 423.609,A -85,B 0,C 180,E1 -16221.752,E2 -16221.752} C_VEL
LIN {X 0,Y 448.143,Z 432.936,A -85,B 0,C 180,E1 -16224.344,E2 -16224.344} C_VEL
LIN {X 0,Y 457.39,Z 446.075,A -85,B 0,C 180,E1 -16227.328,E2 -16227.328} C_VEL
LIN {X 0,Y 467.572,Z 461.659,A -85,B 0,C 180,E1 -16230.204,E2 -16230.204} C_VEL
LIN {X 0,Y 476.832,Z 476.803,A -85,B 0,C 180,E1 -16232.545,E2 -16232.545} C_VEL
LIN {X 0,Y 486.373,Z 493.527,A -85,B 0,C 180,E1 -16234.749,E2 -16234.749} C_VEL
LIN {X 0,Y 487.083,Z 495.289,A -85,B 0,C 180,E1 -16234.917,E2 -16234.917} C_VEL
LIN {X 0,Y 473.187,Z 745.087,A -85,B 0,C 180,E1 -16238.854,E2 -16238.854} C_VEL
LIN {X 0,Y 471.117,Z 771.554,A -85,B 0,C 180,E1 -16239.339,E2 -16239.339} C_VEL
LIN {X 0,Y 468.45,Z 793.432,A -85,B 0,C 180,E1 -16239.867,E2 -16239.867} C_VEL
LIN {X 0,Y 464.436,Z 818.378,A -85,B 0,C 180,E1 -16240.666,E2 -16240.666} C_VEL
LIN {X 0,Y 460.667,Z 837.803,A -85,B 0,C 180,E1 -16241.454,E2 -16241.454} C_VEL
LIN {X 0,Y 455.615,Z 860.692,A -85,B 0,C 180,E1 -16242.584,E2 -16242.584} C_VEL
LIN {X 0,Y 450.208,Z 881.742,A -85,B 0,C 180,E1 -16243.863,E2 -16243.863} C_VEL
LIN {X 0,Y 444.695,Z 901.411,A -85,B 0,C 180,E1 -16245.269,E2 -16245.269} C_VEL
LIN {X 0,Y 438.111,Z 922.871,A -85,B 0,C 180,E1 -16247.106,E2 -16247.106} C_VEL
LIN {X 0,Y 432.585,Z 939.743,A -85,B 0,C 180,E1 -16248.795,E2 -16248.795} C_VEL
LIN {X 0,Y 425.755,Z 959.582,A -85,B 0,C 180,E1 -16251.118,E2 -16251.118} C_VEL
LIN {X 0,Y 420.065,Z 975.509,A -85,B 0,C 180,E1 -16253.312,E2 -16253.312} C_VEL
LIN {X 0,Y 414.175,Z 991.959,A -85,B 0,C 180,E1 -16255.938,E2 -16255.938} C_VEL
LIN {X 0,Y 409.032,Z 1006.203,A -85,B 0,C 180,E1 -16258.622,E2 -16258.622} C_VEL
LIN {X 0,Y 404.256,Z 1020.075,A -85,B 0,C 180,E1 -16261.648,E2 -16261.648} C_VEL
LIN {X 0,Y 400.198,Z 1032.366,A -85,B 0,C 180,E1 -16264.866,E2 -16264.866} C_VEL
LIN {X 0,Y 396.98,Z 1043.425,A -85,B 0,C 180,E1 -16268.269,E2 -16268.269} C_VEL
LIN {X 0,Y 394.684,Z 1052.453,A -85,B 0,C 180,E1 -16271.691,E2 -16271.691} C_VEL
LIN {X 0,Y 393.201,Z 1059.93,A -85,B 0,C 180,E1 -16275.117,E2 -16275.117} C_VEL
LIN {X 0,Y 392.369,Z 1065.631,A -85,B 0,C 180,E1 -16278.535,E2 -16278.535} C_VEL
LIN {X 0,Y 392.048,Z 1069.387,A -85,B 0,C 180,E1 -16281.493,E2 -16281.493} C_VEL
LIN {X 0,Y 391.95,Z 1072.381,A -85,B 0,C 180,E1 -16284.877,E2 -16284.877} C_VEL
LIN {X 0,Y 391.951,Z 1073.728,A -85,B 0,C 180,E1 -16288.246,E2 -16288.246} C_VEL
LIN {X 0,Y 391.962,Z 1073.786,A -85,B 0,C 180,E1 -16291.023,E2 -16291.023} C_VEL
LIN {X 0,Y 391.946,Z 1072.78,A -85,B 0,C 180,E1 -16293.95,E2 -16293.95} C_VEL
LIN {X 0,Y 391.991,Z 1070.094,A -85,B 0,C 180,E1 -16297.475,E2 -16297.475} C_VEL
LIN {X 0,Y 392.226,Z 1066.319,A -85,B 0,C 180,E1 -16300.576,E2 -16300.576} C_VEL
LIN {X 0,Y 392.778,Z 1061.56,A -85,B 0,C 180,E1 -16303.545,E2 -16303.545} C_VEL
LIN {X 0,Y 394.093,Z 1053.874,A -85,B 0,C 180,E1 -16307.269,E2 -16307.269} C_VEL
LIN {X 0,Y 395.874,Z 1045.813,A -85,B 0,C 180,E1 -16310.399,E2 -16310.399} C_VEL
LIN {X 0,Y 398.671,Z 1035.288,A -85,B 0,C 180,E1 -16313.816,E2 -16313.816} C_VEL
LIN {X 0,Y 401.884,Z 1024.381,A -85,B 0,C 180,E1 -16316.765,E2 -16316.765} C_VEL
LIN {X 0,Y 406.125,Z 1011.269,A -85,B 0,C 180,E1 -16319.823,E2 -16319.823} C_VEL
LIN {X 0,Y 410.98,Z 996.617,A -85,B 0,C 180,E1 -16322.691,E2 -16322.691} C_VEL
LIN {X 0,Y 416.102,Z 981.703,A -85,B 0,C 180,E1 -16325.22,E2 -16325.22} C_VEL
LIN {X 0,Y 422.052,Z 964.053,A -85,B 0,C 180,E1 -16327.764,E2 -16327.764} C_VEL
LIN {X 0,Y 427.606,Z 947.296,A -85,B 0,C 180,E1 -16329.844,E2 -16329.844} C_VEL
LIN {X 0,Y 434.076,Z 926.837,A -85,B 0,C 180,E1 -16332.003,E2 -16332.003} C_VEL
LIN {X 0,Y 439.355,Z 909.137,A -85,B 0,C 180,E1 -16333.596,E2 -16333.596} C_VEL
LIN {X 0,Y 445.485,Z 887.007,A -85,B 0,C 180,E1 -16335.291,E2 -16335.291} C_VEL
LIN {X 0,Y 450.401,Z 867.335,A -85,B 0,C 180,E1 -16336.547,E2 -16336.547} C_VEL
LIN {X 0,Y 455.491,Z 844.733,A -85,B 0,C 180,E1 -16337.764,E2 -16337.764} C_VEL
LIN {X 0,Y 459.84,Z 821.771,A -85,B 0,C 180,E1 -16338.747,E2 -16338.747} C_VEL
LIN {X 0,Y 463.636,Z 798.381,A -85,B 0,C 180,E1 -16339.548,E2 -16339.548} C_VEL
LIN {X 0,Y 466.606,Z 774.03,A -85,B 0,C 180,E1 -16340.165,E2 -16340.165} C_VEL
LIN {X 0,Y 468.518,Z 750.577,A -85,B 0,C 180,E1 -16340.615,E2 -16340.615} C_VEL
LIN {X 0,Y 481.73,Z 500.688,A -85,B 0,C 180,E1 -16344.565,E2 -16344.565} C_VEL
LIN {X 0,Y 482.067,Z 491.701,A -85,B 0,C 180,E1 -16344.732,E2 -16344.732} C_VEL
LIN {X 0,Y 472.219,Z 474.079,A -85,B 0,C 180,E1 -16346.85,E2 -16346.85} C_VEL
LIN {X 0,Y 462.43,Z 457.753,A -85,B 0,C 180,E1 -16349.139,E2 -16349.139} C_VEL
LIN {X 0,Y 452.462,Z 442.354,A -85,B 0,C 180,E1 -16351.704,E2 -16351.704} C_VEL
LIN {X 0,Y 445.961,Z 432.998,A -85,B 0,C 180,E1 -16353.537,E2 -16353.537} C_VEL
LIN {X 0,Y 439.102,Z 423.302,A -85,B 0,C 180,E1 -16355.659,E2 -16355.659} C_VEL
LIN {X 0,Y 433.648,Z 416.334,A -85,B 0,C 180,E1 -16357.495,E2 -16357.495} C_VEL
LIN {X 0,Y 429.886,Z 411.664,A -85,B 0,C 180,E1 -16358.868,E2 -16358.868} C_VEL
LIN {X 0,Y 425.512,Z 406.796,A -85,B 0,C 180,E1 -16360.579,E2 -16360.579} C_VEL
LIN {X 0,Y 424.17,Z 404.903,A -85,B 0,C 180,E1 -16361.159,E2 -16361.159} C_VEL
LIN {X 0,Y 420.773,Z 401.5,A -85,B 0,C 180,E1 -16362.649,E2 -16362.649} C_VEL
LIN {X 0,Y 419.067,Z 398.833,A -85,B 0,C 180,E1 -16363.505,E2 -16363.505} C_VEL
LIN {X 0,Y 415.64,Z 396.018,A -85,B 0,C 180,E1 -16365.226,E2 -16365.226} C_VEL
LIN {X 0,Y 413.682,Z 392.463,A -85,B 0,C 180,E1 -16366.44,E2 -16366.44} C_VEL
LIN {X 0,Y 409.982,Z 390.014,A -85,B 0,C 180,E1 -16368.749,E2 -16368.749} C_VEL
LIN {X 0,Y 408.148,Z 386.758,A -85,B 0,C 180,E1 -16370.268,E2 -16370.268} C_VEL
LIN {X 0,Y 407.71,Z 385.774,A -85,B 0,C 180,E1 -16370.685,E2 -16370.685} C_VEL
LIN {X 0,Y 403.812,Z 383.595,A -85,B 0,C 180,E1 -16374.601,E2 -16374.601} C_VEL
LIN {X 0,Y 401.716,Z 379.418,A -85,B 0,C 180,E1 -16380.143,E2 -16380.143} C_VEL
LIN {X 0,Y 401.699,Z 379.301,A -85,B 0,C 180,E1 -16381.997,E2 -16381.997} C_VEL
LIN {X 0,Y 402.926,Z 382.497,A -85,B 0,C 180,E1 -16386.412,E2 -16386.412} C_VEL
LIN {X 0,Y 406.71,Z 385.47,A -85,B 0,C 180,E1 -16390.912,E2 -16390.912} C_VEL
LIN {X 0,Y 407.878,Z 386.044,A -85,B 0,C 180,E1 -16391.884,E2 -16391.884} C_VEL
LIN {X 0,Y 409.365,Z 389.184,A -85,B 0,C 180,E1 -16393.202,E2 -16393.202} C_VEL
LIN {X 0,Y 412.3,Z 391.844,A -85,B 0,C 180,E1 -16395.184,E2 -16395.184} C_VEL
LIN {X 0,Y 413.753,Z 392.667,A -85,B 0,C 180,E1 -16396.028,E2 -16396.028} C_VEL
LIN {X 0,Y 416.055,Z 396.475,A -85,B 0,C 180,E1 -16397.417,E2 -16397.417} C_VEL
LIN {X 0,Y 419.443,Z 399.307,A -85,B 0,C 180,E1 -16399.098,E2 -16399.098} C_VEL
LIN {X 0,Y 422.238,Z 403.299,A -85,B 0,C 180,E1 -16400.444,E2 -16400.444} C_VEL
LIN {X 0,Y 424.839,Z 405.657,A -85,B 0,C 180,E1 -16401.541,E2 -16401.541} C_VEL
LIN {X 0,Y 428.113,Z 409.894,A -85,B 0,C 180,E1 -16402.885,E2 -16402.885} C_VEL
LIN {X 0,Y 430.045,Z 411.854,A -85,B 0,C 180,E1 -16403.609,E2 -16403.609} C_VEL
LIN {X 0,Y 433.924,Z 416.564,A -85,B 0,C 180,E1 -16405.014,E2 -16405.014} C_VEL
LIN {X 0,Y 439.996,Z 424.177,A -85,B 0,C 180,E1 -16407.033,E2 -16407.033} C_VEL
LIN {X 0,Y 444.51,Z 429.966,A -85,B 0,C 180,E1 -16408.415,E2 -16408.415} C_VEL
LIN {X 0,Y 451.641,Z 439.191,A -85,B 0,C 180,E1 -16410.427,E2 -16410.427} C_VEL
LIN {X 0,Y 461.95,Z 453.355,A -85,B 0,C 180,E1 -16413.056,E2 -16413.056} C_VEL
LIN {X 0,Y 473.346,Z 470.153,A -85,B 0,C 180,E1 -16415.663,E2 -16415.663} C_VEL
LIN {X 0,Y 482.433,Z 484.639,A -85,B 0,C 180,E1 -16417.57,E2 -16417.57} C_VEL
LIN {X 0,Y 468.974,Z 736.412,A -85,B 0,C 180,E1 -16421.549,E2 -16421.549} C_VEL
LIN {X 0,Y 467.181,Z 758.449,A -85,B 0,C 180,E1 -16421.983,E2 -16421.983} C_VEL
LIN {X 0,Y 464.301,Z 783.022,A -85,B 0,C 180,E1 -16422.639,E2 -16422.639} C_VEL
LIN {X 0,Y 460.975,Z 804.43,A -85,B 0,C 180,E1 -16423.395,E2 -16423.395} C_VEL
LIN {X 0,Y 457.064,Z 825.889,A -85,B 0,C 180,E1 -16424.328,E2 -16424.328} C_VEL
LIN {X 0,Y 452.059,Z 849.09,A -85,B 0,C 180,E1 -16425.578,E2 -16425.578} C_VEL
LIN {X 0,Y 447.255,Z 868.657,A -85,B 0,C 180,E1 -16426.835,E2 -16426.835} C_VEL
LIN {X 0,Y 441.166,Z 891.084,A -85,B 0,C 180,E1 -16428.562,E2 -16428.562} C_VEL
LIN {X 0,Y 435.995,Z 908.438,A -85,B 0,C 180,E1 -16430.134,E2 -16430.134} C_VEL
LIN {X 0,Y 429.83,Z 928.005,A -85,B 0,C 180,E1 -16432.196,E2 -16432.196} C_VEL
LIN {X 0,Y 424.092,Z 945.022,A -85,B 0,C 180,E1 -16434.313,E2 -16434.313} C_VEL
LIN {X 0,Y 418.144,Z 962.284,A -85,B 0,C 180,E1 -16436.798,E2 -16436.798} C_VEL
LIN {X 0,Y 412.713,Z 977.598,A -85,B 0,C 180,E1 -16439.418,E2 -16439.418} C_VEL
LIN {X 0,Y 407.773,Z 991.832,A -85,B 0,C 180,E1 -16442.232,E2 -16442.232} C_VEL
LIN {X 0,Y 403.388,Z 1004.565,A -85,B 0,C 180,E1 -16445.235,E2 -16445.235} C_VEL
LIN {X 0,Y 399.844,Z 1015.636,A -85,B 0,C 180,E1 -16448.278,E2 -16448.278} C_VEL
LIN {X 0,Y 396.862,Z 1025.775,A -85,B 0,C 180,E1 -16451.643,E2 -16451.643} C_VEL
LIN {X 0,Y 394.876,Z 1033.558,A -85,B 0,C 180,E1 -16454.744,E2 -16454.744} C_VEL
LIN {X 0,Y 393.323,Z 1040.946,A -85,B 0,C 180,E1 -16458.414,E2 -16458.414} C_VEL
LIN {X 0,Y 392.551,Z 1045.732,A -85,B 0,C 180,E1 -16461.504,E2 -16461.504} C_VEL
LIN {X 0,Y 392.145,Z 1049.646,A -85,B 0,C 180,E1 -16464.88,E2 -16464.88} C_VEL
LIN {X 0,Y 391.997,Z 1051.962,A -85,B 0,C 180,E1 -16468.246,E2 -16468.246} C_VEL
LIN {X 0,Y 391.965,Z 1052.864,A -85,B 0,C 180,E1 -16471.023,E2 -16471.023} C_VEL
LIN {X 0,Y 391.973,Z 1052.777,A -85,B 0,C 180,E1 -16474.096,E2 -16474.096} C_VEL
LIN {X 0,Y 392.058,Z 1051.214,A -85,B 0,C 180,E1 -16477.621,E2 -16477.621} C_VEL
LIN {X 0,Y 392.307,Z 1048.524,A -85,B 0,C 180,E1 -16480.723,E2 -16480.723} C_VEL
LIN {X 0,Y 392.861,Z 1044.661,A -85,B 0,C 180,E1 -16483.842,E2 -16483.842} C_VEL
LIN {X 0,Y 393.592,Z 1040.769,A -85,B 0,C 180,E1 -16486.269,E2 -16486.269} C_VEL
LIN {X 0,Y 393.032,Z 1038.922,A -85,B 0,C 180,E1 -16487.364,E2 -16487.364} C_VEL
LIN {X 0,Y 388.297,Z 1033.538,A -85,B 0,C 180,E1 -16490.302,E2 -16490.302} C_VEL
LIN {X 0,Y 388.161,Z 1031.488,A -85,B 0,C 180,E1 -16491.24,E2 -16491.24} C_VEL
LIN {X 0,Y 391.208,Z 1021.724,A -85,B 0,C 180,E1 -16494.943,E2 -16494.943} C_VEL
LIN {X 0,Y 394.53,Z 1012.11,A -85,B 0,C 180,E1 -16497.96,E2 -16497.96} C_VEL
LIN {X 0,Y 399.372,Z 999.124,A -85,B 0,C 180,E1 -16501.383,E2 -16501.383} C_VEL
LIN {X 0,Y 404.183,Z 986.584,A -85,B 0,C 180,E1 -16504.164,E2 -16504.164} C_VEL
LIN {X 0,Y 410.106,Z 971.471,A -85,B 0,C 180,E1 -16507.029,E2 -16507.029} C_VEL
LIN {X 0,Y 416.021,Z 956.003,A -85,B 0,C 180,E1 -16509.51,E2 -16509.51} C_VEL
LIN {X 0,Y 422.663,Z 938.384,A -85,B 0,C 180,E1 -16511.937,E2 -16511.937} C_VEL
LIN {X 0,Y 428.961,Z 920.629,A -85,B 0,C 180,E1 -16513.997,E2 -16513.997} C_VEL
LIN {X 0,Y 435.548,Z 901.209,A -85,B 0,C 180,E1 -16515.935,E2 -16515.935} C_VEL
LIN {X 0,Y 441.835,Z 880.625,A -85,B 0,C 180,E1 -16517.65,E2 -16517.65} C_VEL
LIN {X 0,Y 447.423,Z 860.804,A -85,B 0,C 180,E1 -16519.056,E2 -16519.056} C_VEL
LIN {X 0,Y 453.017,Z 838.232,A -85,B 0,C 180,E1 -16520.381,E2 -16520.381} C_VEL
LIN {X 0,Y 457.191,Z 818.895,A -85,B 0,C 180,E1 -16521.331,E2 -16521.331} C_VEL
LIN {X 0,Y 461.767,Z 793.938,A -85,B 0,C 180,E1 -16522.32,E2 -16522.32} C_VEL
LIN {X 0,Y 464.905,Z 772.264,A -85,B 0,C 180,E1 -16522.986,E2 -16522.986} C_VEL
LIN {X 0,Y 467.655,Z 747.34,A -85,B 0,C 180,E1 -16523.561,E2 -16523.561} C_VEL
LIN {X 0,Y 471.279,Z 687.121,A -85,B 0,C 180,E1 -16524.543,E2 -16524.543} C_VEL
LIN {X 0,Y 482.561,Z 491.611,A -85,B 0,C 180,E1 -16527.645,E2 -16527.645} C_VEL
LIN {X 0,Y 471.614,Z 474.658,A -85,B 0,C 180,E1 -16530.222,E2 -16530.222} C_VEL
LIN {X 0,Y 462.04,Z 460.876,A -85,B 0,C 180,E1 -16532.726,E2 -16532.726} C_VEL
LIN {X 0,Y 454.319,Z 450.447,A -85,B 0,C 180,E1 -16534.968,E2 -16534.968} C_VEL
LIN {X 0,Y 447.642,Z 441.602,A -85,B 0,C 180,E1 -16537.129,E2 -16537.129} C_VEL
LIN {X 0,Y 443.202,Z 436.029,A -85,B 0,C 180,E1 -16538.701,E2 -16538.701} C_VEL
LIN {X 0,Y 439.218,Z 430.987,A -85,B 0,C 180,E1 -16540.241,E2 -16540.241} C_VEL
LIN {X 0,Y 435.448,Z 426.19,A -85,B 0,C 180,E1 -16541.837,E2 -16541.837} C_VEL
LIN {X 0,Y 431.395,Z 421.665,A -85,B 0,C 180,E1 -16543.713,E2 -16543.713} C_VEL
LIN {X 0,Y 430.163,Z 419.832,A -85,B 0,C 180,E1 -16544.357,E2 -16544.357} C_VEL
LIN {X 0,Y 426.685,Z 416.352,A -85,B 0,C 180,E1 -16546.24,E2 -16546.24} C_VEL
LIN {X 0,Y 425.161,Z 413.779,A -85,B 0,C 180,E1 -16547.228,E2 -16547.228} C_VEL
LIN {X 0,Y 421.812,Z 411.007,A -85,B 0,C 180,E1 -16549.483,E2 -16549.483} C_VEL
LIN {X 0,Y 419.877,Z 407.432,A -85,B 0,C 180,E1 -16551.233,E2 -16551.233} C_VEL
LIN {X 0,Y 415.834,Z 404.429,A -85,B 0,C 180,E1 -16556.001,E2 -16556.001} C_VEL
LIN {X 0,Y 414.742,Z 401.753,A -85,B 0,C 180,E1 -16559.862,E2 -16559.862} C_VEL
LIN {X 0,Y 414.717,Z 401.619,A -85,B 0,C 180,E1 -16561.382,E2 -16561.382} C_VEL
LIN {X 0,Y 415.242,Z 403.337,A -85,B 0,C 180,E1 -16564.281,E2 -16564.281} C_VEL
LIN {X 0,Y 419.25,Z 407.195,A -85,B 0,C 180,E1 -16569.888,E2 -16569.888} C_VEL
LIN {X 0,Y 420.088,Z 407.737,A -85,B 0,C 180,E1 -16570.63,E2 -16570.63} C_VEL
LIN {X 0,Y 422.241,Z 411.567,A -85,B 0,C 180,E1 -16572.514,E2 -16572.514} C_VEL
LIN {X 0,Y 425.517,Z 414.256,A -85,B 0,C 180,E1 -16574.667,E2 -16574.667} C_VEL
LIN {X 0,Y 428.154,Z 418.196,A -85,B 0,C 180,E1 -16576.275,E2 -16576.275} C_VEL
LIN {X 0,Y 430.667,Z 420.442,A -85,B 0,C 180,E1 -16577.567,E2 -16577.567} C_VEL
LIN {X 0,Y 434.083,Z 424.878,A -85,B 0,C 180,E1 -16579.232,E2 -16579.232} C_VEL
LIN {X 0,Y 435.806,Z 426.713,A -85,B 0,C 180,E1 -16579.99,E2 -16579.99} C_VEL
LIN {X 0,Y 439.552,Z 431.305,A -85,B 0,C 180,E1 -16581.554,E2 -16581.554} C_VEL
LIN {X 0,Y 446.538,Z 441.039,A -85,B 0,C 180,E1 -16584.191,E2 -16584.191} C_VEL
LIN {X 0,Y 454.673,Z 452.672,A -85,B 0,C 180,E1 -16586.867,E2 -16586.867} C_VEL
LIN {X 0,Y 464.779,Z 468.395,A -85,B 0,C 180,E1 -16589.799,E2 -16589.799} C_VEL
LIN {X 0,Y 473.883,Z 483.545,A -85,B 0,C 180,E1 -16592.158,E2 -16592.158} C_VEL
LIN {X 0,Y 482.418,Z 498.723,A -85,B 0,C 180,E1 -16594.184,E2 -16594.184} C_VEL
LIN {X 0,Y 468.053,Z 748.938,A -85,B 0,C 180,E1 -16598.145,E2 -16598.145} C_VEL
LIN {X 0,Y 465.972,Z 773.134,A -85,B 0,C 180,E1 -16598.604,E2 -16598.604} C_VEL
LIN {X 0,Y 462.858,Z 797.389,A -85,B 0,C 180,E1 -16599.205,E2 -16599.205} C_VEL
LIN {X 0,Y 458.752,Z 821.123,A -85,B 0,C 180,E1 -16600.003,E2 -16600.003} C_VEL
LIN {X 0,Y 454.683,Z 841.259,A -85,B 0,C 180,E1 -16600.844,E2 -16600.844} C_VEL
LIN {X 0,Y 449.116,Z 864.849,A -85,B 0,C 180,E1 -16602.066,E2 -16602.066} C_VEL
LIN {X 0,Y 444.065,Z 883.795,A -85,B 0,C 180,E1 -16603.246,E2 -16603.246} C_VEL
LIN {X 0,Y 437.897,Z 904.941,A -85,B 0,C 180,E1 -16604.802,E2 -16604.802} C_VEL
LIN {X 0,Y 431.615,Z 924.469,A -85,B 0,C 180,E1 -16606.525,E2 -16606.525} C_VEL
LIN {X 0,Y 425.219,Z 943.337,A -85,B 0,C 180,E1 -16608.462,E2 -16608.462} C_VEL
LIN {X 0,Y 418.497,Z 961.862,A -85,B 0,C 180,E1 -16610.725,E2 -16610.725} C_VEL
LIN {X 0,Y 412.462,Z 978.197,A -85,B 0,C 180,E1 -16613.044,E2 -16613.044} C_VEL
LIN {X 0,Y 406.308,Z 994.527,A -85,B 0,C 180,E1 -16615.779,E2 -16615.779} C_VEL
LIN {X 0,Y 401.467,Z 1007.481,A -85,B 0,C 180,E1 -16618.297,E2 -16618.297} C_VEL
LIN {X 0,Y 396.129,Z 1022.244,A -85,B 0,C 180,E1 -16621.671,E2 -16621.671} C_VEL
LIN {X 0,Y 392.382,Z 1033.25,A -85,B 0,C 180,E1 -16624.652,E2 -16624.652} C_VEL
LIN {X 0,Y 388.944,Z 1044.487,A -85,B 0,C 180,E1 -16628.273,E2 -16628.273} C_VEL
LIN {X 0,Y 386.8,Z 1052.635,A -85,B 0,C 180,E1 -16631.46,E2 -16631.46} C_VEL
LIN {X 0,Y 385.198,Z 1060.295,A -85,B 0,C 180,E1 -16635.109,E2 -16635.109} C_VEL
LIN {X 0,Y 384.382,Z 1065.649,A -85,B 0,C 180,E1 -16638.446,E2 -16638.446} C_VEL
LIN {X 0,Y 384.037,Z 1069.516,A -85,B 0,C 180,E1 -16641.616,E2 -16641.616} C_VEL
LIN {X 0,Y 383.949,Z 1072.401,A -85,B 0,C 180,E1 -16645.22,E2 -16645.22} C_VEL
LIN {X 0,Y 383.953,Z 1073.541,A -85,B 0,C 180,E1 -16648.358,E2 -16648.358} C_VEL
LIN {X 0,Y 383.963,Z 1073.547,A -85,B 0,C 180,E1 -16651.194,E2 -16651.194} C_VEL
LIN {X 0,Y 383.948,Z 1072.419,A -85,B 0,C 180,E1 -16654.331,E2 -16654.331} C_VEL
LIN {X 0,Y 384.004,Z 1069.534,A -85,B 0,C 180,E1 -16657.932,E2 -16657.932} C_VEL
LIN {X 0,Y 384.28,Z 1065.866,A -85,B 0,C 180,E1 -16660.95,E2 -16660.95} C_VEL
LIN {X 0,Y 384.979,Z 1060.531,A -85,B 0,C 180,E1 -16664.285,E2 -16664.285} C_VEL
LIN {X 0,Y 386.406,Z 1052.891,A -85,B 0,C 180,E1 -16667.935,E2 -16667.935} C_VEL
LIN {X 0,Y 388.362,Z 1044.717,A -85,B 0,C 180,E1 -16671.128,E2 -16671.128} C_VEL
LIN {X 0,Y 391.549,Z 1033.43,A -85,B 0,C 180,E1 -16674.759,E2 -16674.759} C_VEL
LIN {X 0,Y 394.875,Z 1022.921,A -85,B 0,C 180,E1 -16677.606,E2 -16677.606} C_VEL
LIN {X 0,Y 399.705,Z 1008.63,A -85,B 0,C 180,E1 -16680.902,E2 -16680.902} C_VEL
LIN {X 0,Y 404.296,Z 995.515,A -85,B 0,C 180,E1 -16683.471,E2 -16683.471} C_VEL
LIN {X 0,Y 409.981,Z 979.623,A -85,B 0,C 180,E1 -16686.172,E2 -16686.172} C_VEL
LIN {X 0,Y 415.936,Z 962.527,A -85,B 0,C 180,E1 -16688.621,E2 -16688.621} C_VEL
LIN {X 0,Y 422.291,Z 944.111,A -85,B 0,C 180,E1 -16690.896,E2 -16690.896} C_VEL
LIN {X 0,Y 428.466,Z 924.968,A -85,B 0,C 180,E1 -16692.881,E2 -16692.881} C_VEL
LIN {X 0,Y 434.363,Z 905.758,A -85,B 0,C 180,E1 -16694.596,E2 -16694.596} C_VEL
LIN {X 0,Y 440.427,Z 884.078,A -85,B 0,C 180,E1 -16696.215,E2 -16696.215} C_VEL
LIN {X 0,Y 445.338,Z 864.832,A -85,B 0,C 180,E1 -16697.429,E2 -16697.429} C_VEL
LIN {X 0,Y 450.75,Z 840.786,A -85,B 0,C 180,E1 -16698.684,E2 -16698.684} C_VEL
LIN {X 0,Y 454.679,Z 820.431,A -85,B 0,C 180,E1 -16699.543,E2 -16699.543} C_VEL
LIN {X 0,Y 458.627,Z 796.402,A -85,B 0,C 180,E1 -16700.353,E2 -16700.353} C_VEL
LIN {X 0,Y 461.517,Z 772.743,A -85,B 0,C 180,E1 -16700.943,E2 -16700.943} C_VEL
LIN {X 0,Y 463.533,Z 747.792,A -85,B 0,C 180,E1 -16701.417,E2 -16701.417} C_VEL
LIN {X 0,Y 477.171,Z 497.629,A -85,B 0,C 180,E1 -16705.388,E2 -16705.388} C_VEL
LIN {X 0,Y 477.14,Z 495.37,A -85,B 0,C 180,E1 -16705.45,E2 -16705.45} C_VEL
LIN {X 0,Y 468.133,Z 479.157,A -85,B 0,C 180,E1 -16707.453,E2 -16707.453} C_VEL
LIN {X 0,Y 458.488,Z 462.849,A -85,B 0,C 180,E1 -16709.786,E2 -16709.786} C_VEL
LIN {X 0,Y 448.517,Z 447.367,A -85,B 0,C 180,E1 -16712.446,E2 -16712.446} C_VEL
LIN {X 0,Y 440.843,Z 436.152,A -85,B 0,C 180,E1 -16714.724,E2 -16714.724} C_VEL
LIN {X 0,Y 435.436,Z 428.576,A -85,B 0,C 180,E1 -16716.485,E2 -16716.485} C_VEL
LIN {X 0,Y 431.436,Z 423.529,A -85,B 0,C 180,E1 -16717.876,E2 -16717.876} C_VEL
LIN {X 0,Y 427.082,Z 418.165,A -85,B 0,C 180,E1 -16719.512,E2 -16719.512} C_VEL
LIN {X 0,Y 423.465,Z 413.928,A -85,B 0,C 180,E1 -16720.983,E2 -16720.983} C_VEL
LIN {X 0,Y 422.283,Z 412.371,A -85,B 0,C 180,E1 -16721.501,E2 -16721.501} C_VEL
LIN {X 0,Y 418.833,Z 408.657,A -85,B 0,C 180,E1 -16723.067,E2 -16723.067} C_VEL
LIN {X 0,Y 417.554,Z 406.557,A -85,B 0,C 180,E1 -16723.729,E2 -16723.729} C_VEL
LIN {X 0,Y 414.063,Z 403.556,A -85,B 0,C 180,E1 -16725.526,E2 -16725.526} C_VEL
LIN {X 0,Y 412.008,Z 400.163,A -85,B 0,C 180,E1 -16726.813,E2 -16726.813} C_VEL
LIN {X 0,Y 408.446,Z 397.48,A -85,B 0,C 180,E1 -16729.135,E2 -16729.135} C_VEL
LIN {X 0,Y 406.632,Z 393.911,A -85,B 0,C 180,E1 -16730.731,E2 -16730.731} C_VEL
LIN {X 0,Y 402.105,Z 390.661,A -85,B 0,C 180,E1 -16735.722,E2 -16735.722} C_VEL
LIN {X 0,Y 400.727,Z 387.333,A -85,B 0,C 180,E1 -16740.286,E2 -16740.286} C_VEL
LIN {X 0,Y 400.721,Z 387.274,A -85,B 0,C 180,E1 -16742.002,E2 -16742.002} C_VEL
LIN {X 0,Y 401.95,Z 390.495,A -85,B 0,C 180,E1 -16746.427,E2 -16746.427} C_VEL
LIN {X 0,Y 405.751,Z 393.425,A -85,B 0,C 180,E1 -16750.938,E2 -16750.938} C_VEL
LIN {X 0,Y 406.606,Z 393.952,A -85,B 0,C 180,E1 -16751.669,E2 -16751.669} C_VEL
LIN {X 0,Y 408.39,Z 397.344,A -85,B 0,C 180,E1 -16753.234,E2 -16753.234} C_VEL
LIN {X 0,Y 411.352,Z 399.841,A -85,B 0,C 180,E1 -16755.22,E2 -16755.22} C_VEL
LIN {X 0,Y 412.319,Z 400.519,A -85,B 0,C 180,E1 -16755.796,E2 -16755.796} C_VEL
LIN {X 0,Y 414.954,Z 404.57,A -85,B 0,C 180,E1 -16757.385,E2 -16757.385} C_VEL
LIN {X 0,Y 417.856,Z 407.066,A -85,B 0,C 180,E1 -16758.847,E2 -16758.847} C_VEL
LIN {X 0,Y 420.843,Z 411.141,A -85,B 0,C 180,E1 -16760.297,E2 -16760.297} C_VEL
LIN {X 0,Y 423.031,Z 413.181,A -85,B 0,C 180,E1 -16761.237,E2 -16761.237} C_VEL
LIN {X 0,Y 426.507,Z 417.6,A -85,B 0,C 180,E1 -16762.684,E2 -16762.684} C_VEL
LIN {X 0,Y 428.237,Z 419.511,A -85,B 0,C 180,E1 -16763.35,E2 -16763.35} C_VEL
LIN {X 0,Y 433.3,Z 425.813,A -85,B 0,C 180,E1 -16765.199,E2 -16765.199} C_VEL
LIN {X 0,Y 438.073,Z 431.845,A -85,B 0,C 180,E1 -16766.794,E2 -16766.794} C_VEL
LIN {X 0,Y 444.947,Z 440.653,A -85,B 0,C 180,E1 -16768.892,E2 -16768.892} C_VEL
LIN {X 0,Y 455.338,Z 454.837,A -85,B 0,C 180,E1 -16771.731,E2 -16771.731} C_VEL
LIN {X 0,Y 465.733,Z 470.04,A -85,B 0,C 180,E1 -16774.266,E2 -16774.266} C_VEL
LIN {X 0,Y 476.542,Z 486.919,A -85,B 0,C 180,E1 -16776.652,E2 -16776.652} C_VEL
LIN {X 0,Y 477.491,Z 488.857,A -85,B 0,C 180,E1 -16776.861,E2 -16776.861} C_VEL
LIN {X 0,Y 463.735,Z 737.904,A -85,B 0,C 180,E1 -16780.819,E2 -16780.819} C_VEL
LIN {X 0,Y 461.873,Z 759.795,A -85,B 0,C 180,E1 -16781.258,E2 -16781.258} C_VEL
LIN {X 0,Y 458.681,Z 785.498,A -85,B 0,C 180,E1 -16781.965,E2 -16781.965} C_VEL
LIN {X 0,Y 455.408,Z 805.842,A -85,B 0,C 180,E1 -16782.695,E2 -16782.695} C_VEL
LIN {X 0,Y 451.039,Z 828.996,A -85,B 0,C 180,E1 -16783.723,E2 -16783.723} C_VEL
LIN {X 0,Y 446.157,Z 850.517,A -85,B 0,C 180,E1 -16784.912,E2 -16784.912} C_VEL
LIN {X 0,Y 440.981,Z 870.936,A -85,B 0,C 180,E1 -16786.246,E2 -16786.246} C_VEL
LIN {X 0,Y 434.94,Z 892.259,A -85,B 0,C 180,E1 -16787.923,E2 -16787.923} C_VEL
LIN {X 0,Y 429.623,Z 909.526,A -85,B 0,C 180,E1 -16789.509,E2 -16789.509} C_VEL
LIN {X 0,Y 422.879,Z 930.049,A -85,B 0,C 180,E1 -16791.722,E2 -16791.722} C_VEL
LIN {X 0,Y 417.38,Z 945.825,A -85,B 0,C 180,E1 -16793.721,E2 -16793.721} C_VEL
LIN {X 0,Y 411.365,Z 962.639,A -85,B 0,C 180,E1 -16796.178,E2 -16796.178} C_VEL
LIN {X 0,Y 405.72,Z 977.942,A -85,B 0,C 180,E1 -16798.833,E2 -16798.833} C_VEL
LIN {X 0,Y 400.577,Z 992.163,A -85,B 0,C 180,E1 -16801.689,E2 -16801.689} C_VEL
LIN {X 0,Y 395.997,Z 1004.877,A -85,B 0,C 180,E1 -16804.74,E2 -16804.74} C_VEL
LIN {X 0,Y 392.289,Z 1015.938,A -85,B 0,C 180,E1 -16807.838,E2 -16807.838} C_VEL
LIN {X 0,Y 389.154,Z 1026.06,A -85,B 0,C 180,E1 -16811.266,E2 -16811.266} C_VEL
LIN {X 0,Y 387.063,Z 1033.804,A -85,B 0,C 180,E1 -16814.415,E2 -16814.415} C_VEL
LIN {X 0,Y 385.412,Z 1041.204,A -85,B 0,C 180,E1 -16818.173,E2 -16818.173} C_VEL
LIN {X 0,Y 384.591,Z 1045.982,A -85,B 0,C 180,E1 -16821.327,E2 -16821.327} C_VEL
LIN {X 0,Y 384.16,Z 1049.886,A -85,B 0,C 180,E1 -16824.773,E2 -16824.773} C_VEL
LIN {X 0,Y 384.002,Z 1052.187,A -85,B 0,C 180,E1 -16828.209,E2 -16828.209} C_VEL
LIN {X 0,Y 383.968,Z 1053.081,A -85,B 0,C 180,E1 -16831.045,E2 -16831.045} C_VEL
LIN {X 0,Y 383.976,Z 1052.987,A -85,B 0,C 180,E1 -16834.181,E2 -16834.181} C_VEL
LIN {X 0,Y 384.07,Z 1051.41,A -85,B 0,C 180,E1 -16837.78,E2 -16837.78} C_VEL
LIN {X 0,Y 384.344,Z 1048.714,A -85,B 0,C 180,E1 -16840.948,E2 -16840.948} C_VEL
LIN {X 0,Y 384.981,Z 1044.641,A -85,B 0,C 180,E1 -16844.285,E2 -16844.285} C_VEL
LIN {X 0,Y 386.285,Z 1038.504,A -85,B 0,C 180,E1 -16847.941,E2 -16847.941} C_VEL
LIN {X 0,Y 388.096,Z 1031.703,A -85,B 0,C 180,E1 -16851.147,E2 -16851.147} C_VEL
LIN {X 0,Y 388.161,Z 1031.488,A -85,B 0,C 180,E1 -16851.24,E2 -16851.24} C_VEL
LIN {X 0,Y 387.959,Z 1029.057,A -85,B 0,C 180,E1 -16852.328,E2 -16852.328} C_VEL
LIN {X 0,Y 384.255,Z 1022.305,A -85,B 0,C 180,E1 -16855.268,E2 -16855.268} C_VEL
LIN {X 0,Y 384.449,Z 1019.742,A -85,B 0,C 180,E1 -16856.188,E2 -16856.188} C_VEL
LIN {X 0,Y 388.656,Z 1008.562,A -85,B 0,C 180,E1 -16859.601,E2 -16859.601} C_VEL
LIN {X 0,Y 393.297,Z 996.716,A -85,B 0,C 180,E1 -16862.614,E2 -16862.614} C_VEL
LIN {X 0,Y 398.824,Z 983.196,A -85,B 0,C 180,E1 -16865.566,E2 -16865.566} C_VEL
LIN {X 0,Y 404.831,Z 968.184,A -85,B 0,C 180,E1 -16868.312,E2 -16868.312} C_VEL
LIN {X 0,Y 411.291,Z 952.107,A -85,B 0,C 180,E1 -16870.841,E2 -16870.841} C_VEL
LIN {X 0,Y 417.998,Z 934.542,A -85,B 0,C 180,E1 -16873.168,E2 -16873.168} C_VEL
LIN {X 0,Y 423.977,Z 918.218,A -85,B 0,C 180,E1 -16875.032,E2 -16875.032} C_VEL
LIN {X 0,Y 431.284,Z 896.797,A -85,B 0,C 180,E1 -16877.106,E2 -16877.106} C_VEL
LIN {X 0,Y 437.077,Z 878.257,A -85,B 0,C 180,E1 -16878.621,E2 -16878.621} C_VEL
LIN {X 0,Y 443.573,Z 855.296,A -85,B 0,C 180,E1 -16880.194,E2 -16880.194} C_VEL
LIN {X 0,Y 448.409,Z 835.821,A -85,B 0,C 180,E1 -16881.302,E2 -16881.302} C_VEL
LIN {X 0,Y 453.294,Z 813.528,A -85,B 0,C 180,E1 -16882.363,E2 -16882.363} C_VEL
LIN {X 0,Y 457.351,Z 790.629,A -85,B 0,C 180,E1 -16883.22,E2 -16883.22} C_VEL
LIN {X 0,Y 460.472,Z 769.119,A -85,B 0,C 180,E1 -16883.86,E2 -16883.86} C_VEL
LIN {X 0,Y 463.129,Z 743.445,A -85,B 0,C 180,E1 -16884.419,E2 -16884.419} C_VEL
LIN {X 0,Y 477.157,Z 509.888,A -85,B 0,C 180,E1 -16888.146,E2 -16888.146} C_VEL
LIN {X 0,Y 477.927,Z 495.802,A -85,B 0,C 180,E1 -16888.386,E2 -16888.386} C_VEL
LIN {X 0,Y 467.87,Z 480.108,A -85,B 0,C 180,E1 -16890.839,E2 -16890.839} C_VEL
LIN {X 0,Y 458.806,Z 466.914,A -85,B 0,C 180,E1 -16893.289,E2 -16893.289} C_VEL
LIN {X 0,Y 449.89,Z 454.557,A -85,B 0,C 180,E1 -16896.001,E2 -16896.001} C_VEL
LIN {X 0,Y 441.733,Z 443.923,A -85,B 0,C 180,E1 -16898.836,E2 -16898.836} C_VEL
LIN {X 0,Y 437.158,Z 438.224,A -85,B 0,C 180,E1 -16900.631,E2 -16900.631} C_VEL
LIN {X 0,Y 432.967,Z 432.988,A -85,B 0,C 180,E1 -16902.46,E2 -16902.46} C_VEL
LIN {X 0,Y 429.53,Z 428.825,A -85,B 0,C 180,E1 -16904.126,E2 -16904.126} C_VEL
LIN {X 0,Y 428.429,Z 427.355,A -85,B 0,C 180,E1 -16904.709,E2 -16904.709} C_VEL
LIN {X 0,Y 424.952,Z 423.571,A -85,B 0,C 180,E1 -16906.668,E2 -16906.668} C_VEL
LIN {X 0,Y 423.763,Z 421.546,A -85,B 0,C 180,E1 -16907.462,E2 -16907.462} C_VEL
LIN {X 0,Y 420.329,Z 418.472,A -85,B 0,C 180,E1 -16909.861,E2 -16909.861} C_VEL
